   IF Activate = CmdResponseType.CommandActivated THEN
	 CASE Axis OF
		AxisSelectType.Az:
			IF Management.ErrorStatus.errAzimuth=0 THEN
				b_activate_Az:=1;
				b_deactivate_Az:=0;
			ELSE 
				Activate := CmdResponseType.CommandFailed;
			END_IF
		AxisSelectType.El:
			IF Management.ErrorStatus.errElevation=0 THEN
				 b_activate_el:=1;
				 b_deactivate_El:=0;
			ELSE 
				Activate := CmdResponseType.CommandFailed;
			END_IF;
		AxisSelectType.Fi:
			IF Management.ErrorStatus.errFeedIndexer=0 THEN
				 b_activate_fi:=1;
				 b_deactivate_Fi:=0;
			ELSE 
				Activate := CmdResponseType.CommandFailed;
			END_IF;
		AxisSelectType.AzEl:
			IF Management.ErrorStatus.errAzimuth=0 AND Management.ErrorStatus.errElevation=0  THEN
				b_activate_Az:=1;
				b_deactivate_Az:=0;
				b_activate_el:=1;
				b_deactivate_el:=0;
			//	b_SCC_enable_off:=FALSE;
			//	b_SCC_enable_on:=TRUE; 
			ELSE 
				Activate := CmdResponseType.CommandFailed;
			END_IF;
		ELSE 
			//Activate := CmdResponseType.ParameterOutOfRange;
		END_CASE
   END_IF
ELSE 
	Activate := CmdResponseType.NoCmdAuth;
END_IF
CommandArbiter.Status.AxisSelect:=Axis;
CommandArbiter.Status.LastCmdResponse:=Activate;
END_METHOD

METHOD DeActivate : UINT
VAR_INPUT
	SessionID: UINT;
	Axis: UINT;
END_VAR
VAR_OUTPUT
	
END_VAR
VAR
END_VAR
CASE CommandArbiter.Status.DscCmdAuthority OF                    // Check that corerct user is issueing a command
	LMC: IF SessionID= CommandArbiter.Lmc_ID THEN
			DeActivate:= CmdResponseType.CommandActivated;
         END_IF
			
	EGUI: IF SessionID= CommandArbiter.Egui_ID THEN
			DeActivate:= CmdResponseType.CommandActivated;
          END_IF		
ELSE 
     DeActivate:= CmdResponseType.NoCmdAuth;
     Command_Arbiter_error:=1;	
END_CASE

IF DeActivate = CmdResponseType.CommandActivated THEN       // Check Dish State
	Command_Arbiter_error:=0;
	CASE Management.Status.DscState OF 
		DSCStateType.StartUp:
		 	DeActivate := CmdResponseType.CommandRejected;
		DSCStateType.Standby:
		 	DeActivate := CmdResponseType.CommandActivated;
		DSCStateType.Locked:
		 	DeActivate := CmdResponseType.DishLocked;
		DSCStateType.Stowed:
		 	DeActivate :=CmdResponseType.Stowed;
		DSCStateType.Locked_Stowed:
		 	DeActivate := CmdResponseType.DishLocked; 
		DSCStateType.Activating :
		 	DeActivate := CmdResponseType.CommandActivated;
		DSCStateType.Deactivating :
		 	DeActivate := CmdResponseType.CommandActivated;
		DSCStateType.Standstill :
		 	DeActivate := CmdResponseType.CommandActivated;
		DSCStateType.Stopping :
		 	DeActivate := CmdResponseType.CommandActivated;
		DSCStateType.Slew :
		 	DeActivate := CmdResponseType.CommandActivated;
		DSCStateType.Jog :
		 	DeActivate := CmdResponseType.CommandActivated;
		DSCStateType.Track :
		 	DeActivate := CmdResponseType.CommandActivated;
	END_CASE

   IF DeActivate = CmdResponseType.CommandActivated THEN     //Deactivate Axis
	 CASE Axis OF
		AxisSelectType.Az:
		   		b_deactivate_Az:=1;                      //Ladder logic checks for motion and stops axis before deactivating              				
				b_activate_Az:=0;             
		AxisSelectType.El:
		    	b_deactivate_El:=1;
				b_activate_el:=0;
		AxisSelectType.Fi:
		    	b_deactivate_Fi:=1;
	    		b_activate_fi:=0;
		AxisSelectType.AzEl:
		    	b_deactivate_Az:=1;
				b_deactivate_El:=1;	
				b_activate_Az:=0;
				b_activate_el:=0;
	ELSE 
		DeActivate := CmdResponseType.ParameterOutOfRange;
	END_CASE
   END_IF
ELSE 
   DeActivate:= CmdResponseType.NoCmdAuth;
END_IF
CommandArbiter.Status.LastCmdResponse:=DeActivate;
END_METHOD

METHOD Move2Band : UINT
VAR_INPUT
	SessionID : UINT;
	Band :UINT;
END_VAR
CASE CommandArbiter.Status.DscCmdAuthority OF                    // Check that correct user is issueing a command
	LMC: IF SessionID= CommandArbiter.Lmc_ID THEN
			Move2Band:= CmdResponseType.CommandActivated;
     	 END_IF
			
	EGUI: IF SessionID= CommandArbiter.Egui_ID THEN
			Move2Band:= CmdResponseType.CommandActivated;
    	  END_IF		
ELSE 
     Move2Band:= CmdResponseType.NoCmdAuth;
     Command_Arbiter_error:=1;	
END_CASE

IF Move2Band = CmdResponseType.CommandActivated THEN // Check Dish State to see if move is possible
	Command_Arbiter_error:=0;
	IF  Management.ErrorStatus.errGeneral=0 AND Management.WarningStatus.waMngmnt =0 THEN  
		CASE Management.Status.DscState OF 
			 DscStateType.Locked:        Move2Band:=CmdResponseType.DishLocked;
			 DscStateType.Locked_Stowed: Move2Band:=CmdResponseType.DishLocked;
			 DscStateType.Standstill:    Move2Band:=CmdResponseType.CommandActivated;
		     DscStateType.Standby:       Move2Band:=CmdResponseType.CommandActivated;
			 DscStateType.Stowed:	     Move2Band:=CmdResponseType.CommandActivated;
			 DscStateType.Slew:  		 Move2Band:=CmdResponseType.CommandActivated;
			 DscStateType.Track:  		 Move2Band:=CmdResponseType.CommandActivated;
			 DscStateType.Activating:	 Move2Band:=CmdResponseType.CommandActivated;
			 DscStateType.Deactivating:	 Move2Band:=CmdResponseType.CommandActivated;
			 DscStateType.Stopping:		 Move2Band:=CmdResponseType.CommandActivated;
			
		ELSE
		     Move2Band:=CmdResponseType.CommandRejected;
		     Command_Arbiter_error:=1;
		END_CASE	
   		CASE Band OF   // get band position
	 		Bandtype.Optical: r_goto_Fi := LREAL_TO_REAL(gc_r_band_optical - r_pos_fi_v); 
                              FeedIndexer.Status.p_Set:= gc_r_band_optical;   
     		Bandtype.Band_1:  r_goto_Fi := LREAL_TO_REAL(gc_r_band_1 - r_pos_fi_v);
							  FeedIndexer.Status.p_Set:= gc_r_band_1;   
	 		Bandtype.Band_2:  r_goto_Fi := LREAL_TO_REAL(gc_r_band_2 - r_pos_fi_v);
							  FeedIndexer.Status.p_Set:= gc_r_band_2;   
	 		Bandtype.Band_3:  r_goto_Fi := LREAL_TO_REAL(gc_r_band_3 - r_pos_fi_v);
						      FeedIndexer.Status.p_Set:= gc_r_band_3;   
	 		Bandtype.Band_4:  r_goto_Fi := LREAL_TO_REAL(gc_r_band_4 - r_pos_fi_v);
							  FeedIndexer.Status.p_Set:= gc_r_band_4;   
	 		Bandtype.Band_5a: r_goto_Fi := LREAL_TO_REAL(gc_r_band_5a - r_pos_fi_v);
							  FeedIndexer.Status.p_Set:= gc_r_band_5a;   
	 		Bandtype.Band_5b: r_goto_Fi := LREAL_TO_REAL(gc_r_band_5b - r_pos_fi_v);
							  FeedIndexer.Status.p_Set:= gc_r_band_5b;   
	 		Bandtype.Band_6:  r_goto_Fi := LREAL_TO_REAL(gc_r_band_6 - r_pos_fi_v);
							  FeedIndexer.Status.p_Set:= gc_r_band_6;
;   
		END_CASE
	
		IF Move2Band = CmdResponseType.CommandActivated THEN  
			b_activate_Fi:=1;
			b_deactivate_Fi:=0;
			r_goto_v_Fi:= r_vel_max_Fi; 
			b_stop_Fi:= FALSE;
			b_start_goto_Fi:= TRUE;
			b_Move2Band_deactivate:= TRUE;
			Move2Band:=CmdResponseType.CommandActivated;
		ELSE 
			Move2Band:=CmdResponseType.ParameterOutOfRange;
		END_IF             			
							
	ELSE
		Move2Band:=CmdResponseType.CommandRejected;
		Command_Arbiter_error:=1;
	END_IF
END_IF

						

CommandArbiter.Status.LastCmdResponse:=Move2Band;
END_METHOD

METHOD Reset : UINT
VAR_INPUT
	SessionID: UINT;
	Axis: UINT;
END_VAR

VAR
	
END_VAR
CASE CommandArbiter.Status.DscCmdAuthority OF                    // Check that corerct user is issueing a command
	LMC: IF SessionID= CommandArbiter.Lmc_ID THEN
			Reset:= CmdResponseType.CommandActivated;
     	 END_IF
			
	EGUI: IF SessionID= CommandArbiter.Egui_ID THEN
			Reset:= CmdResponseType.CommandActivated;
    	  END_IF		
ELSE 
     Reset:= CmdResponseType.NoCmdAuth;
     Command_Arbiter_error:=1;	
END_CASE

IF Reset = CmdResponseType.CommandActivated THEN
	Command_Arbiter_error:=0;
	CASE Management.Status.DscState OF 
		DSCStateType.StartUp:
		 	Reset := CmdResponseType.CommandActivated;
		DSCStateType.Standby:
		 	Reset := CmdResponseType.CommandActivated;
		DSCStateType.Locked:
		 	Reset := CmdResponseType.CommandActivated;
		DSCStateType.Stowed:
		 	Reset :=CmdResponseType.CommandActivated;
		DSCStateType.Locked_Stowed:
		 	Reset := CmdResponseType.CommandActivated;
		DSCStateType.Activating :
		 	Reset := CmdResponseType.CommandRejected;
		DSCStateType.Deactivating :
		 	Reset := CmdResponseType.CommandRejected;
		DSCStateType.Standstill :
		 	Reset := CmdResponseType.CommandRejected;
		DSCStateType.Stopping :
		 	Reset := CmdResponseType.CommandRejected;
		DSCStateType.Slew :
		 	Reset := CmdResponseType.CommandRejected;
		DSCStateType.Jog :
		 	Reset := CmdResponseType.CommandRejected;
		DSCStateType.Track :
		 	Reset := CmdResponseType.CommandRejected;
	END_CASE

	IF Reset = CmdResponseType.CommandActivated THEN
		CASE Axis OF
			AxisSelectType.Az: b_clear_err_Az:= 1;
			AxisSelectType.El: b_clear_err_El:= 1;
			AxisSelectType.Fi: b_clear_err_Fi:= 1;
			AxisSelectType.AzEl: b_clear_err_Az:= 1;
								 b_clear_err_El:= 1;
			AxisSelectType.Unknown: b_clear_err:= 1;
		ELSE
			Reset := CmdResponseType.ParameterOutOfRange;
		END_CASE
	END_IF 
ELSE 
	 Reset:= CmdResponseType.NoCmdAuth;

END_IF

CommandArbiter.Status.LastCmdResponse:=Reset;
END_METHOD

METHOD SetOnSourceThreshold : Uint
VAR_INPUT
	SessionID :UINT;
	OnSourceThreshold : LREAL;
    ThresholdTimePeriod : LREAL;
END_VAR
CASE CommandArbiter.Status.DscCmdAuthority OF                    // Check that corerct user is issueing a command
	LMC: IF SessionID= CommandArbiter.Lmc_ID THEN
			SetOnSourceThreshold:= CmdResponseType.CommandActivated;
     	 END_IF
			
	EGUI: IF SessionID= CommandArbiter.Egui_ID THEN
			SetOnSourceThreshold:= CmdResponseType.CommandActivated;
    	  END_IF		
ELSE 
     SetOnSourceThreshold:= CmdResponseType.NoCmdAuth;
     Command_Arbiter_error:=1;	
END_CASE

IF SetOnSourceThreshold = CmdResponseType.CommandActivated THEN
	IF (OnSourceThreshold > 0 AND Onsourcethreshold <=20) OR ( ThresholdTimePeriod > 0 AND ThresholdTimePeriod <=10) THEN
		Tracking.Status.OnSourceThreshold:= OnSourceThreshold;
		Tracking.Status.ThresholdTimePeriod:=ThresholdTimePeriod;
		 t_onsource_dev_filt:=LREAL_TO_TIME(ThresholdTimePeriod*1000);
	    command_Arbiter_error:=0;
	ELSE
		SetOnSourceThreshold:= CmdResponseType.ParameterOutOfRange;
		Command_Arbiter_error:=1;
	END_IF
	
ELSE 
	 SetOnSourceThreshold:= CmdResponseType.CommandFailed;
	  Command_Arbiter_error:=1;
END_IF

CommandArbiter.Status.LastCmdResponse:=SetOnSourceThreshold;
END_METHOD

METHOD SetPowerMode : UINT (* Command to set the power mode *)
VAR_INPUT
	SessionID: UINT; (*Seesion ID*)
    LowPowerOn: BOOL:= FALSE; (* True = Low Power mode On *)
    PowerLimKw: LREAL:=10; (* Maximum Power limit in High power Mode *)

END_VAR
CASE CommandArbiter.Status.DscCmdAuthority OF                    // Check that correct user is issueing a command
	LMC: IF SessionID= CommandArbiter.Lmc_ID THEN
			SetPowerMode:= CmdResponseType.CommandActivated;
     	 END_IF
			
	EGUI: IF SessionID= CommandArbiter.Egui_ID THEN
			SetPowerMode:= CmdResponseType.CommandActivated;
    	  END_IF		
ELSE 
     SetPowerMode:= CmdResponseType.NoCmdAuth;
     Command_Arbiter_error:=1;	
END_CASE

IF SetPowerMode = CmdResponseType.CommandActivated THEN       // Check Dish State
	Command_Arbiter_error:=0;
	CASE Management.Status.DscState OF 
		DSCStateType.StartUp:
		 	SetPowerMode := CmdResponseType.CommandRejected;
		DSCStateType.Standby:
		 	SetPowerMode := CmdResponseType.CommandActivated;
		DSCStateType.Locked:
		 	SetPowerMode := CmdResponseType.CommandActivated;
		DSCStateType.Stowed:
		 	SetPowerMode :=CmdResponseType.CommandActivated;
		DSCStateType.Locked_Stowed:
		 	SetPowerMode := CmdResponseType.CommandActivated;
		DSCStateType.Activating :
		 	SetPowerMode := CmdResponseType.CommandActivated;
		DSCStateType.Deactivating :
		 	SetPowerMode := CmdResponseType.CommandActivated;
		DSCStateType.Standstill :
		 	SetPowerMode := CmdResponseType.CommandActivated;
		DSCStateType.Stopping :
		 	SetPowerMode := CmdResponseType.CommandActivated;
		DSCStateType.Slew :
		 	SetPowerMode := CmdResponseType.CommandActivated;
		DSCStateType.Jog :
		 	SetPowerMode := CmdResponseType.CommandActivated;
		DSCStateType.Track :
		 	SetPowerMode := CmdResponseType.CommandActivated;
	END_CASE
END_IF

IF SetPowerMode = CmdResponseType.CommandActivated THEN
	//SetPowerMode := CmdResponseType.NotImplemented;
	IF LowPowerOn =1 THEN 
		Management.PowerStatus.LowPowerActive:=1;
		IF Azimuth.Status.Active THEN
			b_deactivate_Az:=1;
			b_activate_Az:=0;
		END_IF
		
		IF Elevation.Status.Active THEN
			b_deactivate_El:=1;
			b_activate_El:=0;
		END_IF
		
		IF FeedIndexer.Status.Active THEN
			b_deactivate_Fi:=1;
	    	b_activate_Fi:=0;
		END_IF 
					
	ELSE
		Management.PowerStatus.LowPowerActive:=0;
		r_vel_max_Az:=  gc_r_power_Kv_Az*PowerLimKw;
  		r_vel_max_El:=  gc_r_power_Kv_El*PowerLimKw;
  		r_vel_max_Fi:=  gc_r_power_Kv_Fi*PowerLimKw;
		r_goto_acc_Az:= gc_r_power_Ka_Az*PowerLimKw;
  		r_goto_acc_El:= gc_r_power_Ka_El*PowerLimKw;
  		r_goto_acc_Fi:= gc_r_power_Ka_Fi*PowerLimKw;
  	END_IF
END_IF

CommandArbiter.Status.LastCmdResponse:=SetPowerMode;
END_METHOD

METHOD Slew2AbsSingleAx : UINT
VAR_INPUT
	SessionID: UINT;
	Axis: Uint;
	Position:LREAL;
	Speed:LREAL;
END_VAR

VAR
END_VAR
CASE CommandArbiter.Status.DscCmdAuthority OF                    // Check that correct user is issueing a command
	LMC: IF SessionID= CommandArbiter.Lmc_ID THEN
			Slew2AbsSingleAx:= CmdResponseType.CommandActivated;
     	 END_IF
			
	EGUI: IF SessionID= CommandArbiter.Egui_ID THEN
			Slew2AbsSingleAx:= CmdResponseType.CommandActivated;
    	  END_IF		
ELSE 
     Slew2AbsSingleAx:= CmdResponseType.NoCmdAuth;
     Command_Arbiter_error:=1;	
END_CASE

IF Slew2AbsSingleAx = CmdResponseType.CommandActivated THEN // Dish State to see if move is possible
	Command_Arbiter_error:=0;
	//IF  Management.ErrorStatus.errGeneral=0 AND Management.WarningStatus.waMngmnt =0 THEN   If the Dish has errors that prevent movement then it will not be in a state where it can be moved. 
		CASE Management.Status.DscState OF 
			 DscStateType.Locked:        Slew2AbsSingleAx:=CmdResponseType.DishLocked;
			 DscStateType.Locked_Stowed: Slew2AbsSingleAx:=CmdResponseType.DishLocked;
			 DscStateType.Standstill:    Slew2AbsSingleAx:=CmdResponseType.CommandActivated;
		     DscStateType.Standby:       Slew2AbsSingleAx:=CmdResponseType.CommandActivated;
			 DscStateType.Stowed:	     Slew2AbsSingleAx:=CmdResponseType.Stowed;
		ELSE
		     Slew2AbsSingleAx:=CmdResponseType.CommandRejected;
		     Command_Arbiter_error:=1;
		END_CASE								
	//ELSE
	//	Slew2AbsAx:=CmdResponseType.CommandAborted;
	//	Command_Arbiter_error:=1;
	//END_IF
END_IF
	
IF Slew2AbsSingleAx = CmdResponseType.CommandActivated THEN  // Move selected axis
	b_goto_rel:=FALSE;
	CASE Axis OF 
		AxisSelectType.Az:	
            IF (Position <= gc_r_pos_max_Az) AND (Position>= gc_r_pos_min_Az) AND (Speed <= gc_r_vel_max_Az*6) THEN
           		b_activate_Az:=1;
			    r_goto_Az := LREAL_TO_REAL(Position);
				 IF Speed > r_vel_max_Az THEN    // For power management
					 r_goto_v_Az:= r_vel_max_Az;
				 ELSE
				 	 r_goto_v_Az:= LREAL_TO_REAL(Speed/6); 
				 END_IF
				b_stop_Az:= FALSE;
				b_start_goto_Az:= TRUE;
				Slew2AbsSingleAx:=CmdResponseType.CommandActivated;
				r_write_position_az_out:=Position; // Writeing setpoint positions to Cyclic out put to get P.Set outputs
			ELSE 
				Slew2AbsSingleAx:=CmdResponseType.ParameterOutOfRange;
			END_IF			   
		AxisSelectType.El:
 			IF (Position <= gc_r_pos_max_El) AND (Position>= gc_r_pos_min_El) AND (Speed <= gc_r_vel_max_El*6
) THEN
            	b_activate_el:=1;
				r_goto_El := LREAL_TO_REAL(Position);
				
				 IF Speed > r_vel_max_El THEN    // For power management
					 r_goto_v_El:= r_vel_max_El;
				 ELSE
				 	 r_goto_v_El:= LREAL_TO_REAL(Speed/6); 
				 END_IF
				
				b_stop_El:= FALSE;
				b_start_goto_El:= TRUE;
				Slew2AbsSingleAx:=CmdResponseType.CommandActivated;
				r_write_position_el_out:=Position; // Writeing setpoint positions to Cyclic out put to get P.Set outputs
			ELSE 
				Slew2AbsSingleAx:=CmdResponseType.ParameterOutOfRange;
			END_IF 
					    
		AxisSelectType.FI: 
			IF (Position <= gc_r_pos_max_Fi) AND (Position >= gc_r_pos_min_Fi) AND (Speed<= gc_r_vel_max_Fi*6) THEN
                 b_activate_Fi:=1;
				 r_goto_Fi := LREAL_TO_REAL(Position);
				 IF Speed > r_vel_max_Fi THEN 
					 r_goto_v_Fi:= r_vel_max_Fi;
				 ELSE
				 	 r_goto_v_Fi:= LREAL_TO_REAL(Speed/6); 
				 END_IF
				 b_stop_Fi:= FALSE;
				 b_start_goto_Fi:= TRUE;
				 Slew2AbsSingleAx:=CmdResponseType.CommandActivated;
				 r_write_position_fi_out:=Position; // Writeing setpoint positions to Cyclic out put to get P.Set outputs
		    ELSE 
				 Slew2AbsSingleAx:=CmdResponseType.ParameterOutOfRange;
			END_IF              
 			     									
	ELSE
		Slew2AbsSingleAx:=CmdResponseType.ParameterOutOfRange;
	END_CASE
END_IF

CommandArbiter.Status.LastCmdResponse:=Slew2AbsSingleAx;
END_METHOD

METHOD Slew2AbsAzEl : UINT
VAR_INPUT
	SessionID:UINT;
	Pos_Az:LREAL;
	Pos_El:LREAL;
	Speed_Az:LREAL;
	Speed_El:LREAL;
END_VAR
VAR_OUTPUT
	
END_VAR
VAR
	fb_TON: TON;  
	b_flip: BOOL:=False ;
END_VAR
CASE CommandArbiter.Status.DscCmdAuthority OF                    // Check that correct user is issueing a command
	LMC: IF SessionID= CommandArbiter.Lmc_ID THEN
			Slew2AbsAzEl:= CmdResponseType.CommandActivated;
     	 END_IF
			
	EGUI: IF SessionID= CommandArbiter.Egui_ID THEN
			Slew2AbsAzEl:= CmdResponseType.CommandActivated;
    	  END_IF		
ELSE 
     Slew2AbsAzEl:= CmdResponseType.NoCmdAuth;
     Command_Arbiter_error:=1;	
END_CASE

IF Slew2AbsAzEl = CmdResponseType.CommandActivated THEN // Dish State to see if move is possible
	Command_Arbiter_error:=0;
	//IF  Management.ErrorStatus.errGeneral=0 AND Management.WarningStatus.waMngmnt =0 THEN  (*The Dish in the standby state*)
		CASE Management.Status.DscState OF 
			 DscStateType.Locked:        Slew2AbsAzEl:=CmdResponseType.DishLocked;
			 DscStateType.Locked_Stowed: Slew2AbsAzEl:=CmdResponseType.DishLocked;
			 DscStateType.Standstill:    Slew2AbsAzEl:=CmdResponseType.CommandActivated;
		     DscStateType.Standby:       Slew2AbsAzEl:=CmdResponseType.CommandActivated;
			 DscStateType.Stowed:	     Slew2AbsAzEl:=CmdResponseType.Stowed;
			 DscStateType.Slew:          Slew2AbsAzEl:=CmdResponseType.CommandActivated;
		ELSE
		     Slew2AbsAzEl:=CmdResponseType.CommandRejected;
		     Command_Arbiter_error:=1;
		END_CASE								
	(*ELSE
		Slew2AbsAzEl:=CmdResponseType.CommandAborted;
		Command_Arbiter_error:=1;
	END_IF*)
END_IF
	
IF Slew2AbsAzEl = CmdResponseType.CommandActivated THEN  // Move selected axis
	b_goto_rel:=FALSE;
	IF ((Pos_Az <= gc_r_pos_max_Az) AND (Pos_Az >= gc_r_pos_min_Az) AND( Speed_Az <= gc_r_vel_max_Az*6)) AND ((Pos_El <= gc_r_pos_max_El) AND (Pos_El >= gc_r_pos_min_El) AND ( Speed_El <= gc_r_vel_max_El*6)) THEN
		IF b_activate_Az=0 THEN   // Activate axis if it is in Standby
			b_activate_Az:=1;
		END_IF
		IF b_activate_El=0 THEN // Activate axis if it is in Standby
		   b_activate_El:=1;
		END_IF
    		
		r_goto_Az := LREAL_TO_REAL(Pos_Az);
		r_goto_v_Az:= LREAL_TO_REAL(Speed_Az/6); 
		b_stop_Az:= FALSE;
		r_goto_El := LREAL_TO_REAL(Pos_El);
		r_goto_v_El:= LREAL_TO_REAL(Speed_El/6); 
		b_stop_El:= FALSE;
		
		b_slew_az_el:=TRUE;
		
				
		Slew2AbsAzEl:=CmdResponseType.CommandActivated;	
	ELSE 
		Slew2AbsAzEl:=CmdResponseType.ParameterOutOfRange;
	END_IF			   
END_IF
r_write_position_az_out:=Pos_Az; // Writeing setpoint positions to Cyclic out put to get P.Set outputs
r_write_position_el_out:=Pos_El;
CommandArbiter.Status.LastCmdResponse:=Slew2AbsAzEl;
END_METHOD

METHOD Slew2RelSingleAx : UINT
VAR_INPUT
	SessionID:UINT;
	Axis: UINT;
	Position:LREAL;
	Speed:LREAL;
END_VAR
CASE CommandArbiter.Status.DscCmdAuthority OF                    // Check that correct user is issueing a command
	LMC: IF SessionID= CommandArbiter.Lmc_ID THEN
			Slew2RelSingleAx:= CmdResponseType.CommandActivated;
     	 END_IF
			
	EGUI: IF SessionID= CommandArbiter.Egui_ID THEN
			Slew2RelSingleAx:= CmdResponseType.CommandActivated;
    	  END_IF		
ELSE 
     Slew2RelSingleAx:= CmdResponseType.NoCmdAuth;
     Command_Arbiter_error:=1;	
END_CASE

IF Slew2RelSingleAx = CmdResponseType.CommandActivated THEN // Dish State to see if move is possible
	Command_Arbiter_error:=0;
	//IF  Management.ErrorStatus.errGeneral=0 AND Management.WarningStatus.waMngmnt =0 THEN  (*The Dish in the standby state*)
		CASE Management.Status.DscState OF 
			 DscStateType.Locked:        Slew2RelSingleAx:=CmdResponseType.DishLocked;
			 DscStateType.Locked_Stowed: Slew2RelSingleAx:=CmdResponseType.DishLocked;
			 DscStateType.Standstill:    Slew2RelSingleAx:=CmdResponseType.CommandActivated;
		     DscStateType.Standby:       Slew2RelSingleAx:=CmdResponseType.CommandActivated;
			 DscStateType.Stowed:	     Slew2RelSingleAx:=CmdResponseType.Stowed;
		ELSE
		     Slew2RelSingleAx:=CmdResponseType.CommandRejected;
		     Command_Arbiter_error:=1;
		END_CASE								
(*	ELSE
		Slew2RelAx:=CmdResponseType.CommandAborted;
		Command_Arbiter_error:=1;
	END_IF*)
END_IF
	
IF Slew2RelSingleAx = CmdResponseType.CommandActivated THEN  // Move selected axis
	CASE Axis OF 
		AxisSelectType.Az:	
            IF ((Position + r_pos_az_v) <= gc_r_pos_max_Az) AND ((Position + r_pos_az_v )>= gc_r_pos_min_Az) AND ( Speed <= gc_r_vel_max_Az*6) THEN
           		b_activate_Az:=1;
			    r_goto_Az := LREAL_TO_REAL(Position);
				r_goto_v_Az:= LREAL_TO_REAL(Speed/6); 
				b_stop_Az:= FALSE;
				b_start_goto_Az:= TRUE;
				b_goto_rel:=TRUE;
				Slew2RelSingleAx:=CmdResponseType.CommandActivated;
			ELSE 
				Slew2RelSingleAx:=CmdResponseType.ParameterOutOfRange;
			END_IF			   
		AxisSelectType.El:
 			IF ((Position + r_pos_el_v) <= gc_r_pos_max_El) AND ((Position + r_pos_el_v )>= gc_r_pos_min_El) AND ( Speed <= gc_r_vel_max_El*6) THEN
            	b_activate_el:=1;
				r_goto_El := LREAL_TO_REAL(Position);
				r_goto_v_El:= LREAL_TO_REAL(Speed/6); 
				b_stop_El:= FALSE;
				b_start_goto_El:= TRUE;
				b_goto_rel:=TRUE;
				Slew2RelSingleAx:=CmdResponseType.CommandActivated;
			ELSE 
				Slew2RelSingleAx:=CmdResponseType.ParameterOutOfRange;
			END_IF 
					    
		AxisSelectType.FI: 
			IF ((Position + r_pos_fi_v) <= gc_r_pos_max_Fi) AND ((Position + r_pos_fi_v )> gc_r_pos_min_Fi) AND ( Speed <= gc_r_vel_max_Fi*6) THEN
                 b_activate_Fi:=1;
				 r_goto_Fi := LREAL_TO_REAL(Position);
				 r_goto_v_Fi:= LREAL_TO_REAL(Speed/6); 
				 b_stop_Fi:= FALSE;
				 b_start_goto_Fi:= TRUE;
				 b_goto_rel:=TRUE;
				 Slew2RelSingleAx:=CmdResponseType.CommandActivated;
		    ELSE 
				 Slew2RelSingleAx:=CmdResponseType.ParameterOutOfRange;
			END_IF              
 			     									
	ELSE
		Slew2RelSingleAx:=CmdResponseType.ParameterOutOfRange;
	END_CASE
	
		
END_IF
CommandArbiter.Status.AxisSelect:=Axis;
CommandArbiter.Status.LastCmdResponse:=Slew2RelSingleAx;
END_METHOD

METHOD Slew2RelAzEl : UINT
VAR_INPUT
	SessionID:UINT;
	Pos_Az:LREAL;
	Pos_El:LREAL;
	Speed_Az:LREAL;
	Speed_El:LREAL;
	
END_VAR
CASE CommandArbiter.Status.DscCmdAuthority OF                    // Check that correct user is issueing a command
	LMC: IF SessionID= CommandArbiter.Lmc_ID THEN
			Slew2RelAzEl:= CmdResponseType.CommandActivated;
     	 END_IF
			
	EGUI: IF SessionID= CommandArbiter.Egui_ID THEN
			Slew2RelAzEl:= CmdResponseType.CommandActivated;
    	  END_IF		
ELSE 
     Slew2RelAzEl:= CmdResponseType.NoCmdAuth;
     Command_Arbiter_error:=1;	
END_CASE

IF Slew2RelAzEl = CmdResponseType.CommandActivated THEN // Dish State to see if move is possible
	Command_Arbiter_error:=0;
	//IF  Management.ErrorStatus.errGeneral=0 AND Management.WarningStatus.waMngmnt =0 THEN  (*The Dish in the standby state*)
		CASE Management.Status.DscState OF 
			 DscStateType.Locked:        Slew2RelAzEl:=CmdResponseType.DishLocked;
			 DscStateType.Locked_Stowed: Slew2RelAzEl:=CmdResponseType.DishLocked;
			 DscStateType.Standstill:    Slew2RelAzEl:=CmdResponseType.CommandActivated;
		     DscStateType.Standby:       Slew2RelAzEl:=CmdResponseType.CommandActivated;
			 DscStateType.Stowed:	     Slew2RelAzEl:=CmdResponseType.Stowed;
		ELSE
		     Slew2RelAzEl:=CmdResponseType.CommandRejected;
		     Command_Arbiter_error:=1;
		END_CASE								
	(*ELSE
		Slew2RelAzEl:=CmdResponseType.CommandAborted;
		Command_Arbiter_error:=1;
	END_IF *)
END_IF
	
IF Slew2RelAzEl = CmdResponseType.CommandActivated THEN  // Move selected axis
	IF (((Pos_Az + r_pos_az_v) <= gc_r_pos_max_Az) AND ((Pos_Az + r_pos_az_v )>= gc_r_pos_min_Az) AND ( Speed_Az <= gc_r_vel_max_Az*6)) AND (((Pos_El + r_pos_el_v) <= gc_r_pos_max_El) AND ((Pos_El + r_pos_el_v )>= gc_r_pos_min_El) AND ( Speed_El <= gc_r_vel_max_El*6)) THEN
    	b_activate_Az:=1;
		r_goto_Az := LREAL_TO_REAL(Pos_Az);
		b_goto_rel:=TRUE;
		r_goto_v_Az:= LREAL_TO_REAL(Speed_Az/6); 
		b_stop_Az:= FALSE;
		b_start_goto_Az:= TRUE;
		b_activate_el:=1;
		r_goto_El := LREAL_TO_REAL(Pos_El);
		r_goto_v_El:= LREAL_TO_REAL(Speed_El/6); 
		b_stop_El:= FALSE;
		b_start_goto_El:= TRUE;
		Slew2RelAzEl:=CmdResponseType.CommandActivated;	
	ELSE 
		Slew2RelAzEl:=CmdResponseType.ParameterOutOfRange;
	END_IF			   
	
END_IF

CommandArbiter.Status.LastCmdResponse:=Slew2RelAzEl;
END_METHOD

METHOD Stop : UINT
VAR_INPUT
	SessionID:Uint;
	Axis: UINT; 
END_VAR
VAR_OUTPUT
	
END_VAR
VAR
	
END_VAR
CASE CommandArbiter.Status.DscCmdAuthority OF                    // Check that corerct user is issueing a command
	LMC: IF SessionID= CommandArbiter.Lmc_ID THEN
			Stop:= CmdResponseType.CommandActivated;
     	 END_IF
			
	EGUI: IF SessionID= CommandArbiter.Egui_ID THEN
			Stop:= CmdResponseType.CommandActivated;
    	  END_IF		
ELSE 
     Stop:= CmdResponseType.NoCmdAuth;
     Command_Arbiter_error:=1;	
END_CASE

IF Stop = CmdResponseType.CommandActivated THEN
	Command_Arbiter_error:=0;
	CASE Management.Status.DscState OF 
		DSCStateType.StartUp:
		 	Stop := CmdResponseType.CommandRejected;
		DSCStateType.Standby:
		 	Stop := CmdResponseType.CommandRejected;
		DSCStateType.Locked:
		 	Stop := CmdResponseType.DishLocked;
		DSCStateType.Stowed:
		 	Stop :=CmdResponseType.Stowed;
		DSCStateType.Locked_Stowed:
		 	Stop := CmdResponseType.DishLocked; 
		DSCStateType.Activating :
		 	Stop := CmdResponseType.CommandRejected;
		DSCStateType.Deactivating :
		 	Stop := CmdResponseType.CommandRejected;
		DSCStateType.Standstill :
		 	Stop := CmdResponseType.CommandActivated;
		DSCStateType.Stopping :
		 	Stop := CmdResponseType.CommandActivated;
		DSCStateType.Slew :
		 	Stop := CmdResponseType.CommandActivated;
		DSCStateType.Jog :
		 	Stop := CmdResponseType.CommandActivated;
		DSCStateType.Track :
		 	Stop := CmdResponseType.CommandActivated;
	END_CASE

	IF Stop = CmdResponseType.CommandActivated THEN
		b_track_on:=0; // In case a track is runnning then stop the track
		CASE Axis OF
			AxisSelectType.Unknown:  // Stops all 
		       b_scc_stop:=1;
			    b_start_goto_Fi:=0;
			AxisSelectType.Az:
			  b_stop_Az:=1;
			  b_start_goto_Az:=0;
			AxisSelectType.El:
			 b_stop_El:=1;
			 b_start_goto_El:=0;
			AxisSelectType.Fi:
			 b_stop_Fi:=1;
			 b_start_goto_Fi:=0;
			AxisSelectType.AzEl:
			  b_scc_stop:=1;
			   b_stop_Az:=1;
			   b_stop_El:=1;
			   b_start_goto_El:=0;
			   b_start_goto_Az:=0;
		ELSE
			Stop := CmdResponseType.ParameterOutOfRange;
		END_CASE
	END_IF 
			
END_IF
CommandArbiter.Status.LastCmdResponse:= Stop;
END_METHOD

METHOD Stow : Uint
VAR_INPUT
	SessionID:UINT;
	StowAction:BOOL;
END_VAR


VAR
	Speed_El: REAL;
	Speed_Az: Real;
END_VAR
CASE CommandArbiter.Status.DscCmdAuthority OF                    // Check that correct user is issueing a command
	LMC: IF SessionID= CommandArbiter.Lmc_ID THEN
			Stow:= CmdResponseType.CommandActivated;
     	 END_IF
			
	EGUI: IF SessionID= CommandArbiter.Egui_ID THEN
			Stow:= CmdResponseType.CommandActivated;
    	  END_IF		
ELSE 
     Stow:= CmdResponseType.NoCmdAuth;
     Command_Arbiter_error:=1;	
END_CASE

IF Stow = CmdResponseType.CommandActivated THEN // Dish State to see if move is possible
	Command_Arbiter_error:=0;
	IF  Management.ErrorStatus.errGeneral=0 AND Management.WarningStatus.waMngmnt =0 THEN  (*The Dish in the standby state*)
		CASE Management.Status.DscState OF 
			 DscStateType.Locked:        Stow:=CmdResponseType.DishLocked;
			 DscStateType.Locked_Stowed: Stow:=CmdResponseType.DishLocked;
			 DscStateType.Standstill:    Stow:=CmdResponseType.CommandActivated;
		     DscStateType.Standby:       Stow:=CmdResponseType.CommandActivated;
			 DscStateType.Slew:          Stow:=CmdResponseType.CommandActivated;
			 DscStateType.Track:         Stow:=CmdResponseType.CommandActivated;
			                              //Stop Track
			 DscStateType.Stowed:	     Stow:=CmdResponseType.CommandActivated;
		ELSE
		     Stow:=CmdResponseType.CommandRejected;
		     Command_Arbiter_error:=1;
		END_CASE								
	ELSE
		Stow:=CmdResponseType.CommandRejected;
		Command_Arbiter_error:=1;
	END_IF
END_IF

IF Stow = CmdResponseType.CommandActivated THEN
	IF StowAction = TRUE THEN 
		b_activate_Az:=1;
		b_activate_el:=1;
		b_stow:=1; 
		
		IF b_UPS_stow THEN 
		   Speed_Az:= gc_UPS_Stow_Az_Speed;
	       Speed_El:=gc_UPS_Stow_El_Speed; 
		ELSE
		   Speed_Az:= gc_r_vel_max_Az;
	       Speed_El:=gc_r_vel_max_El; 
		END_IF
		
		//r_goto_Az := LREAL_TO_REAL(0-r_pos_az_v);
		r_goto_Az :=0;
		r_goto_v_Az:= LREAL_TO_REAL(Speed_Az); 
		r_goto_El := LREAL_TO_REAL(90-r_pos_el_v);
		r_goto_v_El:= LREAL_TO_REAL(Speed_El); 
		
		
        b_stop_Az:= FALSE;
		//b_start_goto_Az:= TRUE;
		b_stop_El:= FALSE;
		//b_start_goto_El:= TRUE;
		
      // Activates ladder logic A_STOW
		b_stow_pin_retract:=0;	
		
		Stow:=CmdResponseType.CommandActivated;	
	ELSIF StowAction = FALSE THEN 
		b_stow_pin_retract:=1 ;
		//b_stow:= 0;	
	END_IF
END_IF
	
r_write_position_az_out:=0; // Writeing setpoint positions to Cyclic out put to get P.Set outputs
r_write_position_el_out:=90;	

CommandArbiter.Status.LastCmdResponse:=Stow;
END_METHOD

METHOD TrackStartDM : UINT
VAR_INPUT
	SessionID:UINT;
	Interpol :UINT; // 0 = Newton 1= Spline
	StartTime : LREAL ;
	
END_VAR
CASE CommandArbiter.Status.DscCmdAuthority OF                    // Check that corerct user is issueing a command
	LMC: IF SessionID= CommandArbiter.Lmc_ID THEN
			TrackStartDM:= CmdResponseType.CommandActivated;
     	 END_IF
			
	EGUI: IF SessionID= CommandArbiter.Egui_ID THEN
			TrackStartDM:= CmdResponseType.CommandActivated;
    	  END_IF		
ELSE 
     TrackStartDM:= CmdResponseType.NoCmdAuth;
     Command_Arbiter_error:=1;	
END_CASE


IF TrackStartDM = CmdResponseType.CommandActivated THEN // Dish State to see if move is possible
	Command_Arbiter_error:=0;
	IF  Management.ErrorStatus.errGeneral=0 AND Management.WarningStatus.waMngmnt =0 THEN  (*The Dish in the standby state*)
		CASE Management.Status.DscState OF 
			 DscStateType.Locked:        TrackStartDM:=CmdResponseType.DishLocked;
			 DscStateType.Locked_Stowed: TrackStartDM:=CmdResponseType.DishLocked;
			 DscStateType.Standstill:    TrackStartDM:=CmdResponseType.CommandActivated;
		     DscStateType.Standby:       TrackStartDM:=CmdResponseType.CommandActivated;
			 DscStateType.Stowed:	     TrackStartDM:=CmdResponseType.Stowed;
		ELSE
		     TrackStartDM:=CmdResponseType.CommandRejected;
		     Command_Arbiter_error:=1;
		END_CASE								
	ELSE
		TrackStartDM:=CmdResponseType.CommandRejected;
		Command_Arbiter_error:=1;
	END_IF
END_IF


IF TrackStartDM= CmdResponseType.CommandActivated AND(StartTime> Time_cds.Status.TAIoffset) THEN
	TrackStartDM:=CmdResponseType.CommandActivated;	
	b_track_start:=1;
	lr_track_start_time:=StartTime;
ELSIF StartTime < 0 THEN  // Times can't be less than zero
	TrackStartDM:=CmdResponseType.ParameterOutOfRange;
ELSE 	
	TrackStartDM:=CmdResponseType.CommandActivated;	
	b_track_start:=1;
	lr_track_start_time:=Time_cds.Status.TAIoffset+0.1; // add 100ms to give enough time to start track. 
END_IF			   



CommandArbiter.Status.LastCmdResponse:=TrackStartDM;
END_METHOD

METHOD TrackStartPolyDM : UINT
VAR_INPUT
	SessionID: UINT;
	TrackId: UINT; 
	Order : UINT;
		
END_VAR
CASE CommandArbiter.Status.DscCmdAuthority OF                    // Check that corerct user is issueing a command
	LMC: IF SessionID= CommandArbiter.Lmc_ID THEN
			TrackStartPolyDM:= CmdResponseType.CommandActivated;
     	 END_IF
			
	EGUI: IF SessionID= CommandArbiter.Egui_ID THEN
			TrackStartPolyDM:= CmdResponseType.CommandActivated;
    	  END_IF		
ELSE 
    TrackStartPolyDM:= CmdResponseType.NoCmdAuth;
     Command_Arbiter_error:=1;	
END_CASE


TrackStartPolyDM:=CmdResponseType.NotImplemented;
CommandArbiter.Status.LastCmdResponse:=TrackStartPolyDM;
END_METHOD

END_FUNCTION_BLOCK

// IndraMotionMlc1/Application/POUs/OPCUA/OPCUA_Method/fb_Pointing
(*{attribute 'opcua.mapping.type' := ''}
{attribute 'opcua.mapping.modeluri' := 'http://skao.int/DS_ICD/'}
{attribute 'opcua.mapping.publicationdate' := '12/14/2023 00:00:00'}
{attribute 'opcua.mapping.nodeid' := 'nsu=http://skao.int/DS_ICD/;i=1014'}*)
FUNCTION_BLOCK fb_Pointing
VAR_INPUT
	Commands: fb_Pointing_Commands;
	Status: PointingStatus_Type;
	AmbTempParameters: AmbTempParam_Type;
	StaticPmParameters: ARRAY [0..7] OF StaticPmParam;
	TiltmeterParameters: TiltmeterParam;
	
	
	
END_VAR
VAR
	TE :LREAL:=0; 
	
END_VAR

END_FUNCTION_BLOCK

// IndraMotionMlc1/Application/POUs/OPCUA/OPCUA_Method/fb_Pointing_Commands
(*{attribute 'opcua.mapping.type' := ''}
{attribute 'opcua.mapping.modeluri' := 'http://skao.int/DS_ICD/'}
{attribute 'opcua.mapping.publicationdate' := '12/14/2023 00:00:00'}
{attribute 'opcua.mapping.nodeid' := 'nsu=http://skao.int/DS_ICD/;i=1014'}*)
FUNCTION_BLOCK fb_Pointing_Commands
VAR_INPUT
	
END_VAR

METHOD AmbTempCorrSetup : UINT

VAR_INPUT
	SessionID:Uint;
	filt_dt:LREAL;
	ambTempParam1:LREAL;
	ambTempParam2:LREAL;
	ambTempParam3:LREAL;
	ambTempParam4:LREAL;
	ambTempParam5:LREAL;
	ambTempParam6:LREAL;
END_VAR
VAR_OUTPUT
	
END_VAR
VAR
END_VAR
IF SessionID = CommandArbiter.Egui_ID AND CommandArbiter.Status.DscCmdAuthority= EGUI THEN
	Command_Arbiter_error:=0;
	IF filt_dt>=0 AND  filt_dt<=1000 THEN         // Only checks if filt_dt is in range
		Pointing.AmbTempParameters.filt_dt:=filt_dt;
		Pointing.AmbTempParameters.ambTempParam1:=ambTempParam1;
		Pointing.AmbTempParameters.ambTempParam2:=ambTempParam2;
		Pointing.AmbTempParameters.ambTempParam3:=ambTempParam3;
		Pointing.AmbTempParameters.ambTempParam4:=ambTempParam4;
		Pointing.AmbTempParameters.ambTempParam5:=ambTempParam5;
		Pointing.AmbTempParameters.ambTempParam6:=ambTempParam6;	
		AmbTempCorrSetup:=CmdResponseType.CommandDone;
	ELSE
		AmbTempCorrSetup:=CmdResponseType.ParameterOutOfRange;		
	END_IF
ELSE
  AmbTempCorrSetup:=CmdResponseType.NoCmdAuth;
Command_Arbiter_error:=1;	
END_IF

CommandArbiter.Status.LastCmdResponse:= AmbTempCorrSetup;
END_METHOD

METHOD PmCorrOnOff : UINT

VAR_INPUT
	SessionID:UINT;
	StaticOn:BOOL;
	TiltOn:UINT;
	AmbTOn:BOOL;
	Band:UINT;
	
END_VAR
VAR_OUTPUT
	
END_VAR
VAR
END_VAR
CASE CommandArbiter.Status.DscCmdAuthority OF                    // Check that corerct user is issueing a command
	LMC: IF SessionID= CommandArbiter.Lmc_ID THEN
			PmCorrOnOff:= CmdResponseType.CommandActivated;
         END_IF
			
	EGUI: IF SessionID= CommandArbiter.Egui_ID THEN
			PmCorrOnOff:= CmdResponseType.CommandActivated;
     	  END_IF		
ELSE 
     PmCorrOnOff:= CmdResponseType.NoCmdAuth;
     Command_Arbiter_error:=1;	
END_CASE

IF PmCorrOnOff = CmdResponseType.CommandActivated THEN 
	IF  Band <8 AND Band >= 0 THEN 
		Command_Arbiter_error:=0;
		Pointing.Status.BandForCorr:=Band;
		PmCorrOnOff:=CmdResponseType.CommandDone;
		IF StaticOn THEN
	    	Pointing.Status.StaticCorrActive:=TRUE;
		ELSE
			Pointing.Status.StaticCorrActive:=FALSE;		
		END_IF
		
		IF AmbTOn THEN
			Pointing.Status.AmbTempCorrActive:=TRUE;
		ELSE
			Pointing.Status.AmbTempCorrActive:=FALSE;	
		END_IF
	
		CASE TiltOn OF
        	0: Pointing.Status.TiltCorrActive:=0;
			   Pointing.Status.TiltOne_On:=0;
			   Pointing.Status.TiltTwo_On:=0;
						
        	1: Pointing.Status.TiltCorrActive:=1;
		   	   Pointing.Status.TiltOne_On:=1;
			   Pointing.Status.TiltTwo_On:=0;
			   
			2: Pointing.Status.TiltCorrActive:=1;
		   	   Pointing.Status.TiltOne_On:=0;
			   Pointing.Status.TiltTwo_On:=1;
   	 	ELSE
			PmCorrOnOff:=CmdResponseType.ParameterOutOfRange;
		END_CASE
	   
	ELSE 
		PmCorrOnOff:=CmdResponseType.ParameterOutOfRange;
	END_IF
END_IF
CommandArbiter.Status.LastTiltOn:=TiltOn;
CommandArbiter.Status.LastCmdResponse:= PmCorrOnOff;
END_METHOD

METHOD StaticPmSetup : UINT
VAR_INPUT
	SessionID:UINT;
	Band:UINT;
	IA:LREAL;
	CA:LREAL;
	NPAE:LREAL;
	AN:LREAL;
	AN0:LREAL;
	AW:LREAL;
	AW0:LREAL;
	ACEC:LREAL;
	ACES:LREAL;
	ABA:LREAL;
	ABphi:LREAL;
	IE:LREAL;
	ECEC: LREAL;
	ECES: LREAL;
	HECE4: LREAL;
	HESE4:LREAL;
	HECE8:LREAL;
	HESE8:LREAL;

END_VAR
VAR_OUTPUT
	
END_VAR
VAR
END_VAR
CASE CommandArbiter.Status.DscCmdAuthority OF                    // Check that corerct user is issueing a command
	LMC: IF SessionID= CommandArbiter.Lmc_ID THEN
			StaticPmSetup:= CmdResponseType.CommandActivated;
         END_IF
			
	EGUI: IF SessionID= CommandArbiter.Egui_ID THEN
			StaticPmSetup:= CmdResponseType.CommandActivated;
     	  END_IF		
ELSE 
     StaticPmSetup:= CmdResponseType.NoCmdAuth;
     Command_Arbiter_error:=1;	
END_CASE



IF StaticPmSetup = CmdResponseType.CommandActivated  THEN
	Command_Arbiter_error:=0;
	IF Band >=0 AND Band <8 THEN
		Pointing.StaticPmParameters[Band].IA:=IA;
		Pointing.StaticPmParameters[Band].CA:=CA;
		Pointing.StaticPmParameters[Band].NPAE:=NPAE;
		Pointing.StaticPmParameters[Band].AN:=AN;
		Pointing.StaticPmParameters[Band].AN0:=AN0;
		Pointing.StaticPmParameters[Band].AW:=AW;
		Pointing.StaticPmParameters[Band].AW0:=AW0;
		Pointing.StaticPmParameters[Band].ACEC:=ACEC;
		Pointing.StaticPmParameters[Band].ACES:=ACES;
		Pointing.StaticPmParameters[Band].ABA:=ABA;
		Pointing.StaticPmParameters[Band].ABphi:=ABphi;
		Pointing.StaticPmParameters[Band].IE:=IE;
		Pointing.StaticPmParameters[Band].ECEC:=ECEC;
		Pointing.StaticPmParameters[Band].ECES:=ECES;
		Pointing.StaticPmParameters[Band].HECE4:=HECE4;
		Pointing.StaticPmParameters[Band].HESE4:=HESE4;
		Pointing.StaticPmParameters[Band].HECE8:=HECE8;
		Pointing.StaticPmParameters[Band].HESE8:=HESE8;
		StaticPmSetup:=CmdResponseType.CommandDone;
	ELSE
   		StaticPmSetup:=CmdResponseType.ParameterOutOfRange;	
	END_IF
ELSE
   StaticPmSetup:=CmdResponseType.NoCmdAuth;	
   Command_Arbiter_error:=1;
END_IF
CommandArbiter.Status.LastCmdResponse:=StaticPmSetup;
END_METHOD

METHOD TiltCalSetup : UINT
VAR_INPUT
	SessionID:Uint;
	TiltmeterPos:UINT;
	Tiltmeter_serial_no:STRING;
	tilt_temp_scale:LREAL;
	x_filt_dt:LREAL;
	x_off:LREAL;
	x_offTC:LREAL;
	x_scale:LREAL;
	x_scaleTC:LREAL;
	x_zero:LREAL;
	x_zeroTC:LREAL;
	y_filt_dt:LREAL;
	y_off:LREAL;
	y_offTC:LREAL;
	y_scale:LREAL;
	y_scaleTC:LREAL;
	y_zero:LREAL;
	y_zeroTC:LREAL;
	
	
END_VAR
VAR_OUTPUT
	
END_VAR
VAR
END_VAR
IF SessionID = CommandArbiter.Egui_ID AND CommandArbiter.Status.DscCmdAuthority = EGUI THEN
	Command_Arbiter_error:=0;
	IF TiltmeterPos=1  THEN
		Pointing.TiltmeterParameters.One.Tiltmeter_serial_no:=Tiltmeter_serial_no;
		Pointing.TiltmeterParameters.One.Tilt_temp_scale:=Tilt_temp_scale;
		Pointing.TiltmeterParameters.One.x_scale:=x_scale;
		Pointing.TiltmeterParameters.One.x_scaleTC:=x_scaleTC;
		Pointing.TiltmeterParameters.One.x_zero:=x_zero;
		Pointing.TiltmeterParameters.One.x_zeroTC:=x_zeroTC;
		Pointing.TiltmeterParameters.One.x_off:=x_off;
		Pointing.TiltmeterParameters.One.x_offTC:=x_offTC;
		Pointing.TiltmeterParameters.One.x_filt_dt:=x_filt_dt;
		Pointing.TiltmeterParameters.One.y_scale:=y_scale;
		Pointing.TiltmeterParameters.One.y_scaleTC:=y_scaleTC;
		Pointing.TiltmeterParameters.One.y_zero:=y_zero;
		Pointing.TiltmeterParameters.One.y_zeroTC:=y_zeroTC;
		Pointing.TiltmeterParameters.One.y_off:=y_off;
		Pointing.TiltmeterParameters.One.y_offTC:=y_offTC;
		Pointing.TiltmeterParameters.One.y_filt_dt:=y_filt_dt;
		TiltCalSetup:=CmdResponseType.CommandDone;
	ELSIF TiltmeterPos=2  THEN
		Pointing.TiltmeterParameters.Two.Tiltmeter_serial_no:=Tiltmeter_serial_no;
		Pointing.TiltmeterParameters.Two.Tilt_temp_scale:=Tilt_temp_scale;
		Pointing.TiltmeterParameters.Two.x_scale:=x_scale;
		Pointing.TiltmeterParameters.Two.x_scaleTC:=x_scaleTC;
		Pointing.TiltmeterParameters.Two.x_zero:=x_zero;
		Pointing.TiltmeterParameters.Two.x_zeroTC:=x_zeroTC;
		Pointing.TiltmeterParameters.Two.x_off:=x_off;
		Pointing.TiltmeterParameters.Two.x_offTC:=x_offTC;
		Pointing.TiltmeterParameters.Two.x_filt_dt:=x_filt_dt;
		Pointing.TiltmeterParameters.Two.y_scale:=y_scale;
		Pointing.TiltmeterParameters.Two.y_scaleTC:=y_scaleTC;
		Pointing.TiltmeterParameters.Two.y_zero:=y_zero;
		Pointing.TiltmeterParameters.Two.y_zeroTC:=y_zeroTC;
		Pointing.TiltmeterParameters.Two.y_off:=y_off;
		Pointing.TiltmeterParameters.Two.y_offTC:=y_offTC;
		Pointing.TiltmeterParameters.Two.y_filt_dt:=y_filt_dt;
		TiltCalSetup:=CmdResponseType.CommandDone;	
	ELSE
		TiltCalSetup:=CmdResponseType.ParameterOutOfRange;		
	END_IF
ELSE
   TiltCalSetup:=CmdResponseType.NoCmdAuth;	
   Command_Arbiter_error:=1;
END_IF

CommandArbiter.Status.LastCmdResponse:=TiltCalSetup;
END_METHOD

END_FUNCTION_BLOCK

// IndraMotionMlc1/Application/POUs/OPCUA/OPCUA_Method/fb_Safety
(*{attribute 'opcua.mapping.type' := ''}
{attribute 'opcua.mapping.modeluri' := 'http://skao.int/DS_ICD/'}
{attribute 'opcua.mapping.publicationdate' := '12/14/2023 00:00:00'}
{attribute 'opcua.mapping.nodeid' := 'nsu=http://skao.int/DS_ICD/;i=1012'}*)
FUNCTION_BLOCK fb_Safety
VAR_INPUT	
	Commands: fb_Safety_Commands;
	Status: SafetyStatus_Type;
	
END_VAR

END_FUNCTION_BLOCK

// IndraMotionMlc1/Application/POUs/OPCUA/OPCUA_Method/fb_Safety_Commands
(*{attribute 'opcua.mapping.type' := ''}
{attribute 'opcua.mapping.modeluri' := 'http://skao.int/DS_ICD/'}
{attribute 'opcua.mapping.publicationdate' := '12/14/2023 00:00:00'}
{attribute 'opcua.mapping.nodeid' := 'nsu=http://skao.int/DS_ICD/;i=1012'}*)
FUNCTION_BLOCK fb_Safety_Commands
VAR_INPUT	
	
	
END_VAR

METHOD InterlockAck :UINT
VAR_INPUT
	SessionID:UINT;	
END_VAR
VAR_OUTPUT
	
END_VAR
VAR
	b_clear_interlock:BOOL;
	
END_VAR
CASE CommandArbiter.Status.DscCmdAuthority OF                    // Check that corerct user is issueing a command
	LMC: IF SessionID = CommandArbiter.Lmc_ID THEN
			InterlockAck:= CmdResponseType.CommandActivated;
         END_IF
			
	EGUI: IF SessionID = CommandArbiter.Egui_ID THEN
		     InterlockAck:= CmdResponseType.CommandActivated;
          END_IF		
ELSE 
     InterlockAck:= CmdResponseType.NoCmdAuth;
     Command_Arbiter_error:=1;	
END_CASE

IF InterlockAck = CmdResponseType.CommandActivated THEN     // Check if the Command can be used in the current dish state
	CASE Management.Status.DscState OF 
		DSCStateType.Locked:
		 	InterlockAck := CmdResponseType.CommandActivated;
		DSCStateType.Locked_Stowed:
		 	InterlockAck := CmdResponseType.CommandActivated;
	ELSE
		InterlockAck := CmdResponseType.CommandFailed;
		Command_Arbiter_error:=1;	
	END_CASE
END_IF

IF InterlockAck = CmdResponseType.CommandActivated THEN   // Clear the interlocks
	Command_Arbiter_error:=0;
  IF  Safety.Status.InterlockClearable THEN
	//b_clear_interlock:=1;
	b_Estop_active:=0;
	b_interlock_active_Az:=0;
	b_interlock_active_El:=0;
	b_interlock_active_Fi:=0;
	Safety.Status.InterlockClearable:=0;
	InterlockAck:=CmdResponseType.CommandDone;		
  ELSE 
	InterlockAck:=CmdResponseType.CommandRejected;
	b_clear_interlock:=0;
  END_IF
END_IF

CommandArbiter.Status.LastCmdResponse:= InterlockAck;
END_METHOD

METHOD MoveStowPin :UINT
VAR_INPUT	
	SessionID: UINT;
	StowPinDeploy:BOOL;
END_VAR
	
VAR_OUTPUT
	
END_VAR
VAR
	Users:STRING;
END_VAR
CASE CommandArbiter.Status.DscCmdAuthority OF                    // Check that corerct user is issueing a command
		
	EGUI: IF SessionID = CommandArbiter.Egui_ID THEN
		     MoveStowPin:= CmdResponseType.CommandActivated;
          ELSE 
			 MoveStowPin:= CmdResponseType.NoCmdAuth;
		  END_IF		
ELSE 
     MoveStowPin:= CmdResponseType.NoCmdAuth;
     Command_Arbiter_error:=1;	
END_CASE

IF MoveStowPin = CmdResponseType.CommandActivated THEN     // Check if the Command can be used in the current dish state
	CASE Management.Status.DscState OF 
		DscStateType.StartUp:
		    MoveStowPin := CmdResponseType.CommandActivated;
		DscStateType.Standstill:
		    MoveStowPin := CmdResponseType.CommandActivated;
		DscStateType.Standby :
			MoveStowPin := CmdResponseType.CommandActivated;
		DSCStateType.Locked:
		 	MoveStowPin := CmdResponseType.DishLocked;
		DSCStateType.Locked_Stowed:
		 	MoveStowPin := CmdResponseType.DishLocked;
		DSCStateType.Stowed	:
		    MoveStowPin := CmdResponseType.CommandActivated;
	ELSE
		MoveStowPin := CmdResponseType.CommandFailed;
		Command_Arbiter_error:=1;	
	END_CASE

END_IF

IF MoveStowPin = CmdResponseType.CommandActivated AND b_stow_lock_allow THEN  // Check that Azimuth is in the correct position 
	Command_Arbiter_error:=0;
			IF StowPinDeploy= TRUE THEN
				IF b_stow_pin_limit_lock  THEN
					MoveStowPin:=CmdResponseType.Stowed;
				ELSE
					b_manual_stow:=1;
					MoveStowPin:=CmdResponseType.CommandActivated;
				END_IF		
			END_IF
	
ELSIF MoveStowPin = CmdResponseType.CommandActivated AND StowPinDeploy= FALSE THEN //Need to be able to retract Stow pin even if Encoders are in incorrect position 
	IF b_stow_pin_limit_unlock  THEN
		MoveStowPin:=CmdResponseType.CommandDone;
	ELSE
		b_manual_stow:=0;
		b_stow_pin_retract:=1;
		MoveStowPin:=CmdResponseType.CommandActivated;
	END_IF		
ELSE 
    MoveStowPin:=CmdResponseType.CommandFailed;			
END_IF		
CommandArbiter.Status.LastCmdResponse:=MoveStowPin;
END_METHOD

END_FUNCTION_BLOCK

// IndraMotionMlc1/Application/POUs/OPCUA/OPCUA_Method/fb_Time_cds
(*{attribute 'opcua.mapping.type' := ''}
{attribute 'opcua.mapping.modeluri' := 'http://skao.int/DS_ICD/'}
{attribute 'opcua.mapping.publicationdate' := '12/14/2023 00:00:00'}
{attribute 'opcua.mapping.nodeid' := 'nsu=http://skao.int/DS_ICD/;i=1023'}*)
FUNCTION_BLOCK fb_Time_cds
VAR_INPUT
	Commands: fb_Time_Commands;
	Status : Time_cdsStatus_Type;
	
END_VAR

END_FUNCTION_BLOCK

// IndraMotionMlc1/Application/POUs/OPCUA/OPCUA_Method/fb_Time_Commands
(*{attribute 'opcua.mapping.type' := ''}
{attribute 'opcua.mapping.modeluri' := 'http://skao.int/DS_ICD/'}
{attribute 'opcua.mapping.publicationdate' := '12/14/2023 00:00:00'}
{attribute 'opcua.mapping.nodeid' := 'nsu=http://skao.int/DS_ICD/;i=1023'}*)
FUNCTION_BLOCK fb_Time_Commands
VAR_INPUT
	
END_VAR

METHOD SetTimeSource : UINT
VAR_INPUT
	SessionID:  UINT;
	DscTimeSyncSource:UINT;
	TimeSourceAddrNTP:STRING;
END_VAR
VAR_OUTPUT
	
END_VAR
IF SessionID = CommandArbiter.Egui_ID AND CommandArbiter.Status.DscCmdAuthority = EGUI THEN
	Command_Arbiter_error:=0;
	CASE DscTimeSyncSource OF 
		DscTimeSyncSourceType.DSC:
			Time_cds.Status.DscTimeSyncSource:= DscTimeSyncSourceType.DSC;
			Source_Timesync:=2;
			SetTimeSource:=CmdResponseType.CommandActivated;
		DscTimeSyncSourceType.NTP:
		    Time_cds.Status.DscTimeSyncSource:= DscTimeSyncSourceType.NTP;
			Source_Timesync:=1;
			IP_Adress_NTP:=TimeSourceAddrNTP;
			SetTimeSource:=CmdResponseType.CommandActivated;
			b_ntp_update_start:=TRUE;
			
		DscTimeSyncSourceType.PTP:
			Time_cds.Status.DscTimeSyncSource:= DscTimeSyncSourceType.PTP;
			Source_Timesync:=0;
			IP_Adress_PTP:=TimeSourceAddrNTP;
			SetTimeSource:=CmdResponseType.CommandActivated;
     ELSE
		 SetTimeSource:=CmdResponseType.ParameterOutOfRange;
	END_CASE
ELSE
   SetTimeSource:=CmdResponseType.NoCmdAuth;
   Command_Arbiter_error:=1;	
END_IF

CommandArbiter.Status.LastCmdResponse:= SetTimeSource;
END_METHOD

END_FUNCTION_BLOCK

// IndraMotionMlc1/Application/POUs/OPCUA/OPCUA_Method/fb_Tracking
(*{attribute 'opcua.mapping.type' := ''}
{attribute 'opcua.mapping.modeluri' := 'http://skao.int/DS_ICD/'}
{attribute 'opcua.mapping.publicationdate' := '12/14/2023 00:00:00'}
{attribute 'opcua.mapping.nodeid' := 'nsu=http://skao.int/DS_ICD/;i=1036'}*)
FUNCTION_BLOCK fb_Tracking
VAR_INPUT
	Commands: fb_Tracking_Commands; 
	Status : TrackingStatus_Type;
	PolyStatus: PolyStatus_type;
	TableStatus: TableStatus_type;
END_VAR

END_FUNCTION_BLOCK

// IndraMotionMlc1/Application/POUs/OPCUA/OPCUA_Method/fb_Tracking_Commands
(*{attribute 'opcua.mapping.type' := ''}
{attribute 'opcua.mapping.modeluri' := 'http://skao.int/DS_ICD/'}
{attribute 'opcua.mapping.publicationdate' := '12/14/2023 00:00:00'}
{attribute 'opcua.mapping.nodeid' := 'nsu=http://skao.int/DS_ICD/;i=1036'}*)
FUNCTION_BLOCK fb_Tracking_Commands
VAR

END_VAR

METHOD TrackLoadStaticOff : Uint
VAR_INPUT
	SessionID:UINT;
	Off_Xel : LREAL;
	Off_El: LREAL;
	
END_VAR
CASE CommandArbiter.Status.DscCmdAuthority OF                    // Check that corerct user is issueing a command
	LMC: IF SessionID= CommandArbiter.Lmc_ID THEN
			TrackLoadStaticOff:= CmdResponseType.CommandActivated;
     	 END_IF
			
	EGUI: IF SessionID= CommandArbiter.Egui_ID THEN
			TrackLoadStaticOff:= CmdResponseType.CommandActivated;
    	  END_IF		
ELSE 
     TrackLoadStaticOff:= CmdResponseType.NoCmdAuth;
     Command_Arbiter_error:=1;	
END_CASE

IF TrackLoadStaticOff = CmdResponseType.CommandActivated THEN 
	IF ABS(Off_El)<= gc_r_El_off_limit AND ABS(Off_Xel)<= gc_r_Xel_off_limit THEN 
	tracking.Status.act_statOffset_value_El:=Off_El;
	tracking.Status.act_statOffset_value_Xel:=Off_Xel;
	ELSE 
		TrackLoadStaticOff:= CmdResponseType.ParameterOutOfRange;
	END_IF
END_IF

CommandArbiter.Status.LastCmdResponse:= TrackLoadStaticOff;
END_METHOD

METHOD TrackLoadTable : UINT
VAR_INPUT
	SessionID:UINT;
	LoadMode :UINT;
	SequenceLength :UINT;
    TaiOffset: ARRAY [1..1000] OF LREAL;
	Azimuth: ARRAY [1..1000] OF LREAL;
	Elevation: ARRAY [1..1000] OF LREAL;
END_VAR

VAR
 i: UINT:=1 ;
 index: UINT:=1 ;
 ValidStart: UINT:=0 ;
END_VAR

CASE CommandArbiter.Status.DscCmdAuthority OF                    // Check that corerct user is issueing a command
	LMC: IF SessionID= CommandArbiter.Lmc_ID THEN
			TrackLoadTable:= CmdResponseType.CommandActivated;
     	 END_IF
			
	EGUI: IF SessionID= CommandArbiter.Egui_ID THEN
			TrackLoadTable:= CmdResponseType.CommandActivated;
    	  END_IF		
ELSE 
     TrackLoadTable:= CmdResponseType.NoCmdAuth;
     Command_Arbiter_error:=1;	
END_CASE

IF TrackLoadTable = CmdResponseType.CommandActivated THEN 
  	IF LoadMode=0 AND(10000-i_num_stack_left) < Sequencelength THEN // Check that there is enough space in the stack.
		TrackLoadTable:= CmdResponseType.CommandFailed;
		
	ELSIF LoadMode=0 AND TaiOffset[SequenceLength] < track_table[i_End].TAIoffset THEN // Check if any point in the loaded table is at the end of the table
		TrackLoadTable:= CmdResponseType.ParameterOutOfRange;
		
	ELSE 
		FOR i:= 1 TO (SequenceLength-1) BY 1 DO    // Check that the time is monotonic 
			IF TaiOffset[i]> (TaiOffset[i+1]) THEN   
				TrackLoadTable:= CmdResponseType.NoOfParametersError;
			END_IF
		END_FOR

		FOR i:= 1 TO SequenceLength BY 1 DO  // Check that the positions are within limits
			IF ((Azimuth[i] > gc_r_pos_max_Az) OR (Azimuth[i] < gc_r_pos_min_Az)) OR ((Elevation[i] > gc_r_pos_max_El) OR (Elevation[i] < gc_r_pos_min_El)) THEN 
				TrackLoadTable:= CmdResponseType.ParameterOutOfRange;
			END_IF
		END_FOR
				
		FOR i:=(SequenceLength-1) TO 1 BY -1 DO    // Check for the time in the Sequence when the future time starts
			IF Time_cds.Status.TAIoffset < (TaiOffset[i+1]+0.1) THEN   
				ValidStart:=i;
			END_IF
		END_FOR
		IF ValidStart < 1 THEN    // Check that table has points in the future 
			TrackLoadTable:= CmdResponseType.ParameterOutOfRange;
		END_IF
	END_IF
END_IF

IF TrackLoadTable = CmdResponseType.CommandActivated THEN 
	CASE LoadMode OF
		  
		0: FOR index:= ValidStart TO SequenceLength BY 1 DO  //Append 
			 IF track_table[i_End].TAIoffset<>0 THEN 
				i_End:=F_I_number(i_End+1);
			 END_IF
			 track_table[i_End].TAIoffset:=TaiOffset[index];
			 track_table[i_End].Azimuth:= Azimuth[index];
			 track_table[i_End].Elevation:= Elevation[index];
			 
		   END_FOR  
           CommandArbiter.Status.LastLoadMode:= LoadMode; 
           
		   
		1:  i_End:= i_Start+1;  // Set the end of the table to the Start to over write the points. 
		                        // Consider adding a blend between the different tables. 
			FOR index:= ValidStart TO SequenceLength BY 1 DO  //New 
			  IF track_table[i_End].TAIoffset<>0 THEN
				 i_End:=F_I_number(i_End+1);
			  END_IF
			  track_table[i_End].TAIoffset:=TaiOffset[index];
			  track_table[i_End].Azimuth:= Azimuth[index];
			  track_table[i_End].Elevation:= Elevation[index];
		    END_FOR            
		   CommandArbiter.Status.LastLoadMode:= LoadMode; 
	       
		2:  i_Start:=1;       // Reset to 1st position of the stack. 
            i_End:= i_Start;  // Set the end of the table to the Start to over write the points. 
		                        // Consider adding a blend between the different tables. 
			FOR index:= ValidStart TO SequenceLength BY 1 DO  //New 
			  IF track_table[i_End].TAIoffset<>0 THEN
				 i_End:=F_I_number(i_End+1);
			  END_IF
			  track_table[i_End].TAIoffset:=TaiOffset[index];
			  track_table[i_End].Azimuth:= Azimuth[index];
			  track_table[i_End].Elevation:= Elevation[index];
		    END_FOR            
	           
	END_CASE;
	TrackLoadTable:= CmdResponseType.CommandActivated; // Reset
	CommandArbiter.Status.LastLoadMode:=LoadMode; 
	Tracking.TableStatus.pts_DataValid:=TRUE;
END_IF;

CommandArbiter.Status.LastCmdResponse:= TrackLoadTable;
END_METHOD

METHOD TrackStart :Uint
VAR_INPUT
	SessionID:UINT;
	Interpol:UINT;
	StartTime:LREAL;
END_VAR
VAR_OUTPUT
	
END_VAR
VAR
	
END_VAR
CASE CommandArbiter.Status.DscCmdAuthority OF                    // Check that corerct user is issueing a command
	LMC: IF SessionID= CommandArbiter.Lmc_ID THEN
			TrackStart:= CmdResponseType.CommandActivated;
     	 END_IF
			
	EGUI: IF SessionID= CommandArbiter.Egui_ID THEN
			TrackStart:= CmdResponseType.CommandActivated;
    	  END_IF		
ELSE 
     TrackStart:= CmdResponseType.NoCmdAuth;
     Command_Arbiter_error:=1;	
END_CASE

IF TrackStart = CmdResponseType.CommandActivated THEN // Dish State to see if move is possible
	Command_Arbiter_error:=0;
	IF  Management.ErrorStatus.errGeneral=0 AND Management.WarningStatus.waMngmnt =0 THEN  (*The Dish in the standby state*)
		CASE Management.Status.DscState OF 
			 DscStateType.Locked:        TrackStart:=CmdResponseType.DishLocked;
			 DscStateType.Locked_Stowed: TrackStart:=CmdResponseType.DishLocked;
			 DscStateType.Standstill:    TrackStart:=CmdResponseType.CommandActivated;
		     DscStateType.Standby:       TrackStart:=CmdResponseType.CommandActivated;
			 DscStateType.Stowed:	     TrackStart:=CmdResponseType.Stowed;
			 DscStateType.Track:         TrackStart:=CmdResponseType.CommandActivated;
		ELSE
		     TrackStart:=CmdResponseType.CommandRejected;
		     Command_Arbiter_error:=1;
		END_CASE								
	ELSE
		TrackStart:=CmdResponseType.CommandRejected;
		Command_Arbiter_error:=1;
	END_IF
END_IF
	
IF TrackStart=CmdResponseType.CommandActivated THEN
	IF StartTime > Time_cds.Status.TAIoffset THEN
		b_activate_Az:=1;
		b_activate_El:=1;	
		b_track_start:=1;
		lr_track_start_time:=StartTime;
	ELSIF StartTime < Time_cds.Status.TAIoffset THEN  // Will start tracking immediately
		b_activate_Az:=1;
		b_activate_El:=1;	
		b_track_start:=1;
		lr_track_start_time:=Time_cds.Status.TAIoffset;
	ELSIF StartTime < 0 THEN 
		TrackStart:=CmdResponseType.ParameterOutOfRange;
	ELSE 	
	//	TrackStart:=CmdResponseType.CommandActivated;
	//	b_activate_Az:=1;
	//	b_activate_El:=1;	
    //b_track_start:=1;
	//	lr_track_start_time:=Time_cds.Status.TAIoffset+0.1; // add 100ms to give enough time to start track. 
	END_IF			   
END_IF

Tracking.TableStatus.pts_Interpol:= Interpol;
CommandArbiter.Status.LastCmdResponse:=TrackStart;
END_METHOD

METHOD TrackStartPoly : UINT

VAR_INPUT
	SessionID:UINT;
	TrackId:  UINT;
	Order : UINT;
END_VAR

VAR
	
END_VAR
// Check Auth
// Check parameters
// Check State
TrackStartPoly := CmdResponseType.NotImplemented;

CommandArbiter.Status.LastCmdResponse:=TrackStartPoly;
END_METHOD

END_FUNCTION_BLOCK

// IndraMotionMlc1/Application/POUs/Panel Function/DANCE_OFF
PROGRAM DANCE_OFF
VAR
	R_TRIG_0: R_TRIG;
	dance_enable: BOOL;
	R_TRIG_1: R_TRIG;
	MC_Power_0: MC_Power;
	MC_MoveAbsolute_0: MC_MoveAbsolute;
	R_TRIG_2: R_TRIG;
	MC_MoveAbsolute_1: MC_MoveAbsolute;
	R_TRIG_3: R_TRIG;
	MC_MoveAbsolute_2: MC_MoveAbsolute;
	R_TRIG_4: R_TRIG;
	dance_step1: BOOL;
	MC_MoveAbsolute_3: MC_MoveAbsolute;
	R_TRIG_5: R_TRIG;
	dance_step2: BOOL;
	MC_MoveAbsolute_4: MC_MoveAbsolute;
	R_TRIG_6: R_TRIG;
	TON_0: TON;
	R_TRIG_7: R_TRIG;
	TON_1: TON;
	dance_step3: BOOL;
	TON_2: TON;
	dance_step4: BOOL;
	MC_MoveAbsolute_5: MC_MoveAbsolute;
	R_TRIG_8: R_TRIG;
	TON_3: TON;
	dance_step5: BOOL;
	MC_MoveAbsolute_6: MC_MoveAbsolute;
	R_TRIG_9: R_TRIG;
	TON_4: TON;
	dance_step6: BOOL;
	MC_MoveAbsolute_7: MC_MoveAbsolute;
	R_TRIG_10: R_TRIG;
	TON_5: TON;
	dance_step7: BOOL;
	R_TRIG_11: R_TRIG;
	dance_step8: BOOL;
	MC_MoveAbsolute_8: MC_MoveAbsolute;
	R_TRIG_12: R_TRIG;
	TON_6: TON;
	F_TRIG_0: F_TRIG;
	TON_7: TON;
	R_TRIG_13: R_TRIG;
	dance_step9: BOOL;
	R_TRIG_14: R_TRIG;
	TON_8: TON;
	TON_9: TON;
	R_TRIG_15: R_TRIG;
	TON_10: TON;
	dance_step10: BOOL;
	TON_11: TON;
END_VAR

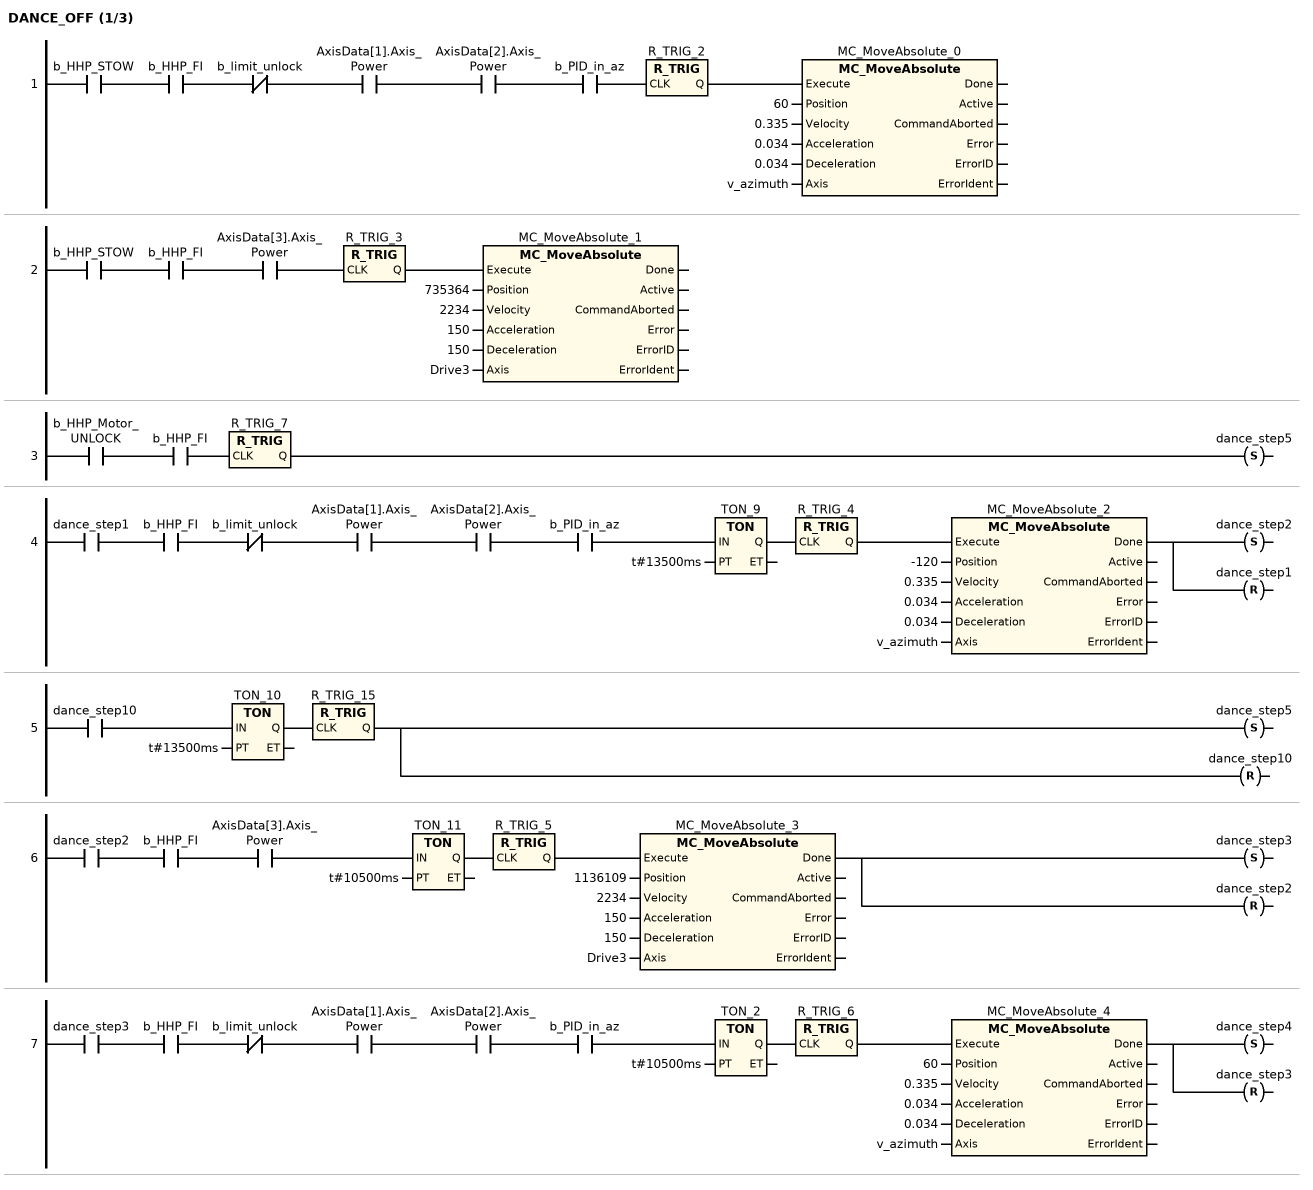
// NETWORK 1
R_TRIG_2(CLK := b_HHP_STOW AND b_HHP_FI AND NOT b_limit_unlock AND AxisData[1].Axis_Power AND AxisData[2].Axis_Power AND b_PID_in_az); // R_TRIG
MC_MoveAbsolute_0(
    Execute := R_TRIG_2.Q,
    Position := 60,
    Velocity := 0.335,
    Acceleration := 0.034,
    Deceleration := 0.034,
    Axis := v_azimuth); // MC_MoveAbsolute

// NETWORK 2
R_TRIG_3(CLK := b_HHP_STOW AND b_HHP_FI AND AxisData[3].Axis_Power); // R_TRIG
MC_MoveAbsolute_1(
    Execute := R_TRIG_3.Q,
    Position := 735364,
    Velocity := 2234,
    Acceleration := 150,
    Deceleration := 150,
    Axis := Drive3); // MC_MoveAbsolute

// NETWORK 3
R_TRIG_7(CLK := b_HHP_Motor_UNLOCK AND b_HHP_FI); // R_TRIG
dance_step5 S= R_TRIG_7.Q;

// NETWORK 4
TON_9(IN := dance_step1 AND b_HHP_FI AND NOT b_limit_unlock AND AxisData[1].Axis_Power AND AxisData[2].Axis_Power AND b_PID_in_az, PT := t#13500ms); // TON
R_TRIG_4(CLK := TON_9.Q); // R_TRIG
MC_MoveAbsolute_2(
    Execute := R_TRIG_4.Q,
    Position := -120,
    Velocity := 0.335,
    Acceleration := 0.034,
    Deceleration := 0.034,
    Axis := v_azimuth); // MC_MoveAbsolute
dance_step2 S= MC_MoveAbsolute_2.Done;
dance_step1 R= MC_MoveAbsolute_2.Done;

// NETWORK 5
TON_10(IN := dance_step10, PT := t#13500ms); // TON
R_TRIG_15(CLK := TON_10.Q); // R_TRIG
dance_step5 S= R_TRIG_15.Q;
dance_step10 R= R_TRIG_15.Q;

// NETWORK 6
TON_11(IN := dance_step2 AND b_HHP_FI AND AxisData[3].Axis_Power, PT := t#10500ms); // TON
R_TRIG_5(CLK := TON_11.Q); // R_TRIG
MC_MoveAbsolute_3(
    Execute := R_TRIG_5.Q,
    Position := 1136109,
    Velocity := 2234,
    Acceleration := 150,
    Deceleration := 150,
    Axis := Drive3); // MC_MoveAbsolute
dance_step3 S= MC_MoveAbsolute_3.Done;
dance_step2 R= MC_MoveAbsolute_3.Done;

// NETWORK 7
TON_2(IN := dance_step3 AND b_HHP_FI AND NOT b_limit_unlock AND AxisData[1].Axis_Power AND AxisData[2].Axis_Power AND b_PID_in_az, PT := t#10500ms); // TON
R_TRIG_6(CLK := TON_2.Q); // R_TRIG
MC_MoveAbsolute_4(
    Execute := R_TRIG_6.Q,
    Position := 60,
    Velocity := 0.335,
    Acceleration := 0.034,
    Deceleration := 0.034,
    Axis := v_azimuth); // MC_MoveAbsolute
dance_step4 S= MC_MoveAbsolute_4.Done;
dance_step3 R= MC_MoveAbsolute_4.Done;

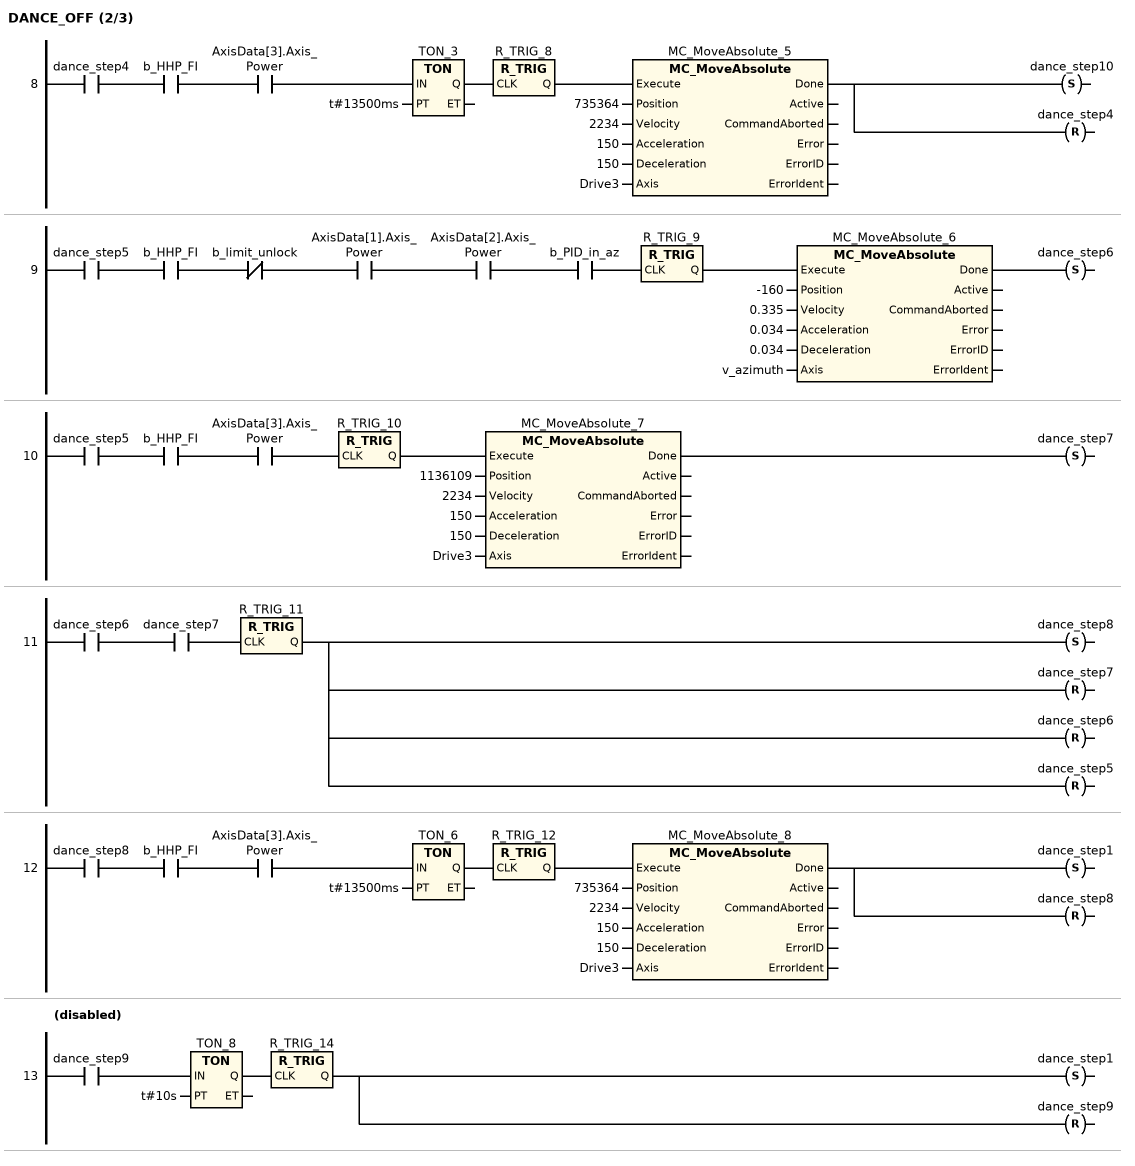
// NETWORK 8
TON_3(IN := dance_step4 AND b_HHP_FI AND AxisData[3].Axis_Power, PT := t#13500ms); // TON
R_TRIG_8(CLK := TON_3.Q); // R_TRIG
MC_MoveAbsolute_5(
    Execute := R_TRIG_8.Q,
    Position := 735364,
    Velocity := 2234,
    Acceleration := 150,
    Deceleration := 150,
    Axis := Drive3); // MC_MoveAbsolute
dance_step10 S= MC_MoveAbsolute_5.Done;
dance_step4 R= MC_MoveAbsolute_5.Done;

// NETWORK 9
R_TRIG_9(CLK := dance_step5 AND b_HHP_FI AND NOT b_limit_unlock AND AxisData[1].Axis_Power AND AxisData[2].Axis_Power AND b_PID_in_az); // R_TRIG
MC_MoveAbsolute_6(
    Execute := R_TRIG_9.Q,
    Position := -160,
    Velocity := 0.335,
    Acceleration := 0.034,
    Deceleration := 0.034,
    Axis := v_azimuth); // MC_MoveAbsolute
dance_step6 S= MC_MoveAbsolute_6.Done;

// NETWORK 10
R_TRIG_10(CLK := dance_step5 AND b_HHP_FI AND AxisData[3].Axis_Power); // R_TRIG
MC_MoveAbsolute_7(
    Execute := R_TRIG_10.Q,
    Position := 1136109,
    Velocity := 2234,
    Acceleration := 150,
    Deceleration := 150,
    Axis := Drive3); // MC_MoveAbsolute
dance_step7 S= MC_MoveAbsolute_7.Done;

// NETWORK 11
R_TRIG_11(CLK := dance_step6 AND dance_step7); // R_TRIG
dance_step8 S= R_TRIG_11.Q;
dance_step7 R= R_TRIG_11.Q;
dance_step6 R= R_TRIG_11.Q;
dance_step5 R= R_TRIG_11.Q;

// NETWORK 12
TON_6(IN := dance_step8 AND b_HHP_FI AND AxisData[3].Axis_Power, PT := t#13500ms); // TON
R_TRIG_12(CLK := TON_6.Q); // R_TRIG
MC_MoveAbsolute_8(
    Execute := R_TRIG_12.Q,
    Position := 735364,
    Velocity := 2234,
    Acceleration := 150,
    Deceleration := 150,
    Axis := Drive3); // MC_MoveAbsolute
dance_step1 S= MC_MoveAbsolute_8.Done;
dance_step8 R= MC_MoveAbsolute_8.Done;

// NETWORK 13 (disabled)
// TON_8(IN := dance_step9, PT := t#10s); // TON
// R_TRIG_14(CLK := TON_8.Q); // R_TRIG
// dance_step1 S= R_TRIG_14.Q;
// dance_step9 R= R_TRIG_14.Q;

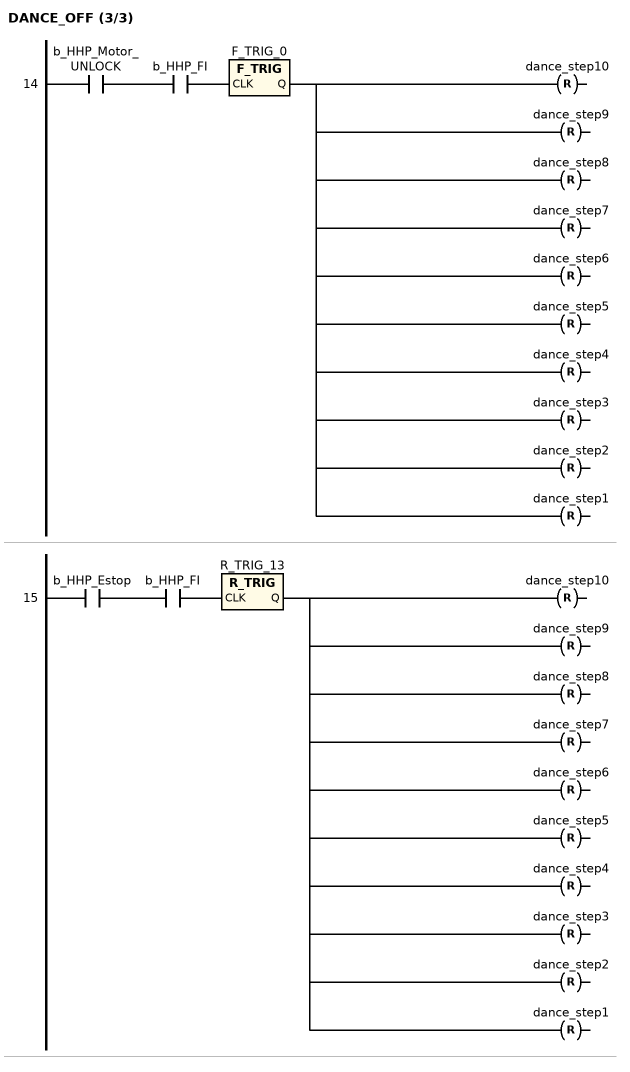
// NETWORK 14
F_TRIG_0(CLK := b_HHP_Motor_UNLOCK AND b_HHP_FI); // F_TRIG
dance_step10 R= F_TRIG_0.Q;
dance_step9 R= F_TRIG_0.Q;
dance_step8 R= F_TRIG_0.Q;
dance_step7 R= F_TRIG_0.Q;
dance_step6 R= F_TRIG_0.Q;
dance_step5 R= F_TRIG_0.Q;
dance_step4 R= F_TRIG_0.Q;
dance_step3 R= F_TRIG_0.Q;
dance_step2 R= F_TRIG_0.Q;
dance_step1 R= F_TRIG_0.Q;

// NETWORK 15
R_TRIG_13(CLK := b_HHP_Estop AND b_HHP_FI); // R_TRIG
dance_step10 R= R_TRIG_13.Q;
dance_step9 R= R_TRIG_13.Q;
dance_step8 R= R_TRIG_13.Q;
dance_step7 R= R_TRIG_13.Q;
dance_step6 R= R_TRIG_13.Q;
dance_step5 R= R_TRIG_13.Q;
dance_step4 R= R_TRIG_13.Q;
dance_step3 R= R_TRIG_13.Q;
dance_step2 R= R_TRIG_13.Q;
dance_step1 R= R_TRIG_13.Q;

END_PROGRAM

// IndraMotionMlc1/Application/POUs/Motion/P_Read_Parameters
(* The program is modified from the program that was built for GSTAT and KSTAT,according to ICD*)
PROGRAM P_Read_Parameters
VAR

(*The function block BLINK generates a pulsating signal.The input consists of ENABLE of the type BOOL, as well as TIMELOW and TIMEHIGH of the type TIME.*)
	fb_blink_diagnos_1: BLINK;
	fb_blink_diagnos_2: BLINK;
	fb_blink_diagnos_3: BLINK;
	fb_blink_diagnos_4: BLINK;
	fb_blink_diagnos_5: BLINK;
	fb_blink_diagnos_6: BLINK;
	fb_blink_diagnos_MLC: BLINK;
(*With the function block "MB_ReadParameter" it is possible to read the current value of a parameter. The return value is DINT*)
	fb_read_brake_1: MB_ReadParameter;
	fb_read_brake_2: MB_ReadParameter;
	fb_read_brake_3: MB_ReadParameter;
	fb_read_brake_4: MB_ReadParameter;
	fb_read_brake_5: MB_ReadParameter;
	fb_read_brake_6: MB_ReadParameter;
(*With the function block "MB_ReadStringParameter" it is possible to read a parameter the operating data of which has the ASCII format (string).*)
	fb_diagnose_1: MB_ReadStringParameter;
	fb_diagnose_2: MB_ReadStringParameter;
	fb_diagnose_3: MB_ReadStringParameter;
	fb_diagnose_4: MB_ReadStringParameter;
	fb_diagnose_5: MB_ReadStringParameter;
	fb_diagnose_6: MB_ReadStringParameter;
	fb_diagnose_MLC: MB_ReadStringParameter;
(*With the function block "MB_ReadRealParameter" it is possible to read the current value of a parameter. The return value is REAL. *)
	FB_readcur1: MB_ReadRealParameter;
	FB_readcur2: MB_ReadRealParameter;
	FB_readcur3: MB_ReadRealParameter;
	FB_readcur4: MB_ReadRealParameter;
	FB_readcur5: MB_ReadRealParameter;
	FB_readcur6: MB_ReadRealParameter;
	fb_temp_1: MB_ReadRealParameter;
	fb_temp_2: MB_ReadRealParameter;
	fb_temp_3: MB_ReadRealParameter;
	fb_temp_4: MB_ReadRealParameter;
	fb_temp_5: MB_ReadRealParameter;
	fb_temp_6: MB_ReadRealParameter;
	fb_read_s189_1: MB_ReadRealParameter;
	fb_read_s189_3: MB_ReadRealParameter;
	fb_read_s189_5: MB_ReadRealParameter;
	FB_readtor1: MB_ReadRealParameter;
	FB_readtor2: MB_ReadRealParameter;
	FB_readtor3: MB_ReadRealParameter;
	FB_readtor4: MB_ReadRealParameter;
	FB_readtor5: MB_ReadRealParameter;
	FB_readtor6: MB_ReadRealParameter;
	FB_temp_1_a: MB_ReadRealParameter;
	FB_temp_2_a: MB_ReadRealParameter;
	FB_temp_3_a: MB_ReadRealParameter;
	FB_temp_4_a: MB_ReadRealParameter;
	FB_temp_5_a: MB_ReadRealParameter;
	FB_temp_6_a: MB_ReadRealParameter;
(*FP_P_0_0539,Holding brake status word *)
	dw_brake_1: DWORD;
	dw_brake_2: DWORD;
	dw_brake_3: DWORD;
	dw_brake_4: DWORD;
	dw_brake_5: DWORD;
	dw_brake_6: DWORD;
(*FP_P_0_0007,Display text of diagnostic message*)
	str_diagnose_MLC: STRING;
	str_diagnose_1: STRING;
	str_diagnose_2: STRING;
	str_diagnose_3: STRING;
	str_diagnose_4: STRING;
	str_diagnose_5: STRING;
	str_diagnose_6: STRING;

(*FP_S_0_0384,Amplifier temperature*)
	r_temp_amp1: REAL;
	r_temp_amp2: REAL;
	r_temp_amp3: REAL;
	r_temp_amp4: REAL;
	r_temp_amp5: REAL;
	r_temp_amp6: REAL;


(*<<<<<<<<<<<<<<<<<<<<<<<<<<<<<<<<<<<<<<<add MLC temperature and operation hour(20100708)>>>>>>>>>>>>>>>>>>>>>>>>>>>>>>>>>>>>>*)
	fb_temp_MLC: MB_ReadRealParameter;
	r_temp_MLC: REAL;(*FP_c_0_0070,Control unit temperature*)
	fb_read_system_status: MB_ReadParameter;
	dw_system_status: DWORD;(*FP_C_0_0023,MC system status,used for temperature warning*)
	fb_read_operation_hour: MB_ReadParameter;

(*the limit for judging whether azimuth following error is too big*)
	r_limit_track_az: REAL;
(*test for limit check*)
	fb_software_limit_1: MB_ReadParameter;
	fb_software_limit_5: MB_ReadParameter;
	fb_software_limit_3: MB_ReadParameter;
	fb_hardware_limit_1: MB_ReadParameter;
	fb_hardware_limit_3: MB_ReadParameter;
	fb_hardware_limit_5: MB_ReadParameter;
	fb_ESTOP_1: MB_ReadParameter;
	fb_ESTOP_3: MB_ReadParameter;
	fb_ESTOP_5: MB_ReadParameter;
	i_software_limit_1: DINT;
	i_software_limit_3: DINT;
	i_software_limit_5: DINT;
	i_hardware_limit_1: DINT;
	i_hardware_limit_3: DINT;
	i_hardware_limit_5: DINT;
	i_ESTOP_1: DINT;
	i_ESTOP_3: DINT;
	i_ESTOP_5: DINT;


	b_azimuth_limit: BOOL;
	b_elevation_limit: BOOL;
	b_FeedIndexer_limit: BOOL;
	fb_readpar_speed_1: MB_ReadRealParameter;
	fb_readpar_speed_3: MB_ReadRealParameter;
	fb_readpar_speed_5: MB_ReadRealParameter;
	
	str_concat: ARRAY[1..40] OF STRING(1500);(*数组及其类型的定义*)	
	Counter: INT;
	FB_readmotorencoder1: MB_ReadRealParameter;
	FB_readmotorencoder2: MB_ReadRealParameter;
	FB_readmotorencoder3: MB_ReadRealParameter;
	FB_readmotorencoder4: MB_ReadRealParameter;
	FB_readmotorencoder5: MB_ReadRealParameter;
	FB_readmotorencoder6: MB_ReadRealParameter;
	r_motorencoder_6: REAL;
	r_motorencoder_5: REAL;
	r_motorencoder_4: REAL;
	r_motorencoder_3: REAL;
	r_motorencoder_2: REAL;
	r_motorencoder_1: REAL;
	
	(*the status word for GSTAT*)
	
	status_1:DWORD;
	status_2:DWORD;
	status_3:DWORD;
	status_4:DWORD;
	status_5:DWORD;
	status_6:DWORD;
	fb_diagnose_111: MB_ReadParameter;
	str_diagnose_11: DWORD;
	fb_blink_diagnos_11: BLINK;
	fb_diagnose_11: MB_ReadrealParameter;
	str_diagnose_111: REAL;
	fb_readpar_speed_2: MB_ReadRealParameter;
	fb_readpar_speed_4: MB_ReadRealParameter;
	fb_readpar_speed_6: MB_ReadRealParameter;
	
	ReadAxisPshape: ARRAY[1..5] OF MB_ReadlrealParameter;
	ReadAxisVact: ARRAY[1..5] OF MB_ReadlrealParameter;
	ReadAxisVshape: ARRAY[1..5] OF MB_ReadlrealParameter;

	conut_i: INT;
	b_PID_in_FI: BOOL;
	b_limit_cw_FI: BOOL;
	b_limit_ccw_FI: BOOL;
	b_limit_final_FI: BOOL;
	fb_readpar_pos_cmd_1: MB_ReadRealParameter;
END_VAR

P_Read_Parameters.A_Read_Parameter();

status_code1:=LEFT(str_diagnose_1,5);
status_code2:=LEFT(str_diagnose_2,5);
status_code3:=LEFT(str_diagnose_3,5);
status_code4:=LEFT(str_diagnose_4,5);
status_code5:=LEFT(str_diagnose_5,5);
status_code6:=LEFT(str_diagnose_6,5);

FOR  conut_i:=1 TO 5 BY 1 DO
ReadAxisPshape[conut_i](
	Enable:=axisdata[1].Axis_Inbb , 
	Done=> , 
	Active=> , 
	Error=> , 
	ErrorID=> , 
	ErrorIdent=> , 
	ParameterNumber:=FP_P_0_0434 , 
	Value=>P_shape_value[conut_i] , 
	Axis:=AxRef[conut_i] );
	
ReadAxisVshape[conut_i](
	Enable:=axisdata[1].Axis_Inbb , 
	Done=> , 
	Active=> , 
	Error=> , 
	ErrorID=> , 
	ErrorIdent=> , 
	ParameterNumber:=FP_P_0_0434 , 
	Value=>V_shape_value[conut_i] , 
	Axis:=AxRef[conut_i] );
	
ReadAxisVact[conut_i](
	Enable:=axisdata[1].Axis_Inbb , 
	Done=> , 
	Active=> , 
	Error=> , 
	ErrorID=> , 
	ErrorIdent=> , 
	ParameterNumber:=FP_S_0_0040 , 
	Value=>V_act_value[conut_i] , 
	Axis:=AxRef[conut_i] );
END_FOR
(*
(*<<<<<<<<<<<<<<<<<<<<<<<<<<<<<master_status>>>>>>>>>>>>>>>>>>>>>>>>>>>>>>>>>>>>>>>>>>>>>>>>>>>>>>>*)
master_status.0:=axisdata[1].Axis_InAb;
IF b_remote_on=TRUE THEN
	master_status.1:=0;
ELSE
	master_status.1:=1;
END_IF
IF b_DSdoor_Estop  THEN
	master_status.2:=1;
ELSE
	master_status.2:=0;
END_IF

IF ABS(axisdata[3].rActualPosition_i-90)<0.02 THEN
	master_status.3:=1;
ELSE
	master_status.3:=0;
END_IF
	master_status.4:=(axisdata[1].Axis_Error OR axisdata[2].Axis_Error OR axisdata[3].Axis_Error OR axisdata[4].Axis_Error OR axisdata[5].Axis_Error OR axisdata[6].Axis_Error);
	master_status.5:=b_stow_pin_limit_unlock;
	master_status.6:=b_stow_pin_limit_lock;
	
IF i_num_stack_left>9500 THEN
		master_status.7:=0;
	ELSE IF i_num_stack_left<1500 THEN
		master_status.7:=1;	
	END_IF
		
END_IF

IF b_remote_on_run AND b_track_on THEN
	master_status.9:=0;
	master_status.8:=1;
ELSIF b_remote_on_run AND b_Track_Pause = TRUE THEN
	master_status.9:=1;
	master_status.8:=0;
ELSIF b_remote_on_run AND b_Track_Pause = FALSE  AND b_track_on = FALSE THEN
	master_status.9:=0;
	master_status.8:=0;
ELSE
 	master_status.9:=1;
	master_status.8:=1;
END_IF

IF 	b_encoder_ok_az	AND b_encoder_ok_FI THEN
	master_status.10:=1;
	master_status.11:=1;
ELSIF b_encoder_ok_az =FALSE AND b_encoder_ok_FI THEN
	master_status.10:=0;
	master_status.11:=1;
ELSIF b_encoder_ok_az  AND b_encoder_ok_FI=FALSE THEN
	master_status.10:=1;
	master_status.11:=0;
ELSE
	master_status.10:=0;
	master_status.11:=0;		
END_IF

IF b_remote_on_run THEN
	master_status.12:=1;
ELSE
	master_status.12:=0;
END_IF
	
IF b_remote_on_run THEN
	master_status.12:=1;
ELSE
	master_status.12:=0;
END_IF

IF b_permit_new_file THEN
	master_status.13:=1;
ELSE
	master_status.13:=0;
END_IF

(*<<<<<<<<<<<<<<<<<<<<<<<<<<<<<status_1>>>>>>>>>>>>>>>>>>>>>>>>>>>>>>>>>>>>>>>>>>>>>>>>>>>>>>>*)
status_1.0:=axisdata[1].Axis_InAb;
status_1.1:=b_PID_in_az;
status_1.2:=dw_brake_1.0;
status_1.3:=b_limit_cw_az;
status_1.4:=b_limit_ccw_az;
status_1.5:=(b_limit_final_cw_az OR b_limit_final_ccw_az);
status_1.6:=axisdata[1].Axis_Error;

(*<<<<<<<<<<<<<<<<<<<<<<<<<<<<<status_2>>>>>>>>>>>>>>>>>>>>>>>>>>>>>>>>>>>>>>>>>>>>>>>>>>>>>>>*)
status_2.0:=axisdata[2].Axis_InAb;
status_2.1:=b_PID_in_az;
status_2.2:=dw_brake_2.0;
status_2.3:=b_limit_cw_az;
status_2.4:=b_limit_ccw_az;
status_2.5:=(b_limit_final_cw_az OR b_limit_final_ccw_az);
status_2.6:=axisdata[2].Axis_Error;

(*<<<<<<<<<<<<<<<<<<<<<<<<<<<<<status_3>>>>>>>>>>>>>>>>>>>>>>>>>>>>>>>>>>>>>>>>>>>>>>>>>>>>>>>*)
status_3.0:=axisdata[3].Axis_InAb;
status_3.1:=b_PID_in_el;
status_3.2:=dw_brake_3.0;
status_3.3:=b_limit_cw_el;
status_3.4:=b_limit_ccw_el;
status_3.5:=(b_limit_final_cw_el OR b_limit_final_ccw_el) ;
status_3.6:=axisdata[3].Axis_Error;

(*<<<<<<<<<<<<<<<<<<<<<<<<<<<<<status_4>>>>>>>>>>>>>>>>>>>>>>>>>>>>>>>>>>>>>>>>>>>>>>>>>>>>>>>*)
status_4.0:=axisdata[4].Axis_InAb;
status_4.1:=b_PID_in_el;
status_4.2:=dw_brake_4.0;
status_4.3:=b_limit_cw_el;
status_4.4:=b_limit_ccw_el;
status_4.5:=(b_limit_final_cw_el OR b_limit_final_ccw_el); 
status_4.6:=axisdata[4].Axis_Error;

(*<<<<<<<<<<<<<<<<<<<<<<<<<<<<<status_5>>>>>>>>>>>>>>>>>>>>>>>>>>>>>>>>>>>>>>>>>>>>>>>>>>>>>>>*)
status_5.0:=axisdata[5].Axis_InAb;
status_5.1:=b_PID_in_FI;
status_5.2:=dw_brake_5.0;
status_5.3:=b_limit_cw_FI;
status_5.4:=b_limit_ccw_FI;
status_5.5:=b_limit_final_FI;
status_5.6:=axisdata[5].Axis_Error;

(*<<<<<<<<<<<<<<<<<<<<<<<<<<<<<status_6>>>>>>>>>>>>>>>>>>>>>>>>>>>>>>>>>>>>>>>>>>>>>>>>>>>>>>>*)
status_6.0:=axisdata[6].Axis_InAb;
status_6.1:=b_PID_in_FI;
status_6.2:=dw_brake_6.0;
status_6.3:=b_limit_cw_FI;
status_6.4:=b_limit_ccw_FI;
status_6.5:=b_limit_final_FI;
status_6.6:=axisdata[6].Axis_Error;


(*
(*<<<<<<<<<<<<<<<<<<<<<<<<<<<<<status_2>>>>>>>>>>>>>>>>>>>>>>>>>>>>>>>>>>>>>>>>>>>>>>>>>>>>>>>*)
status_2.0:=NOT(axisdata[2].Axis_InAb);
status_2.1:=axisdata[2].Axis_Error;
status_2.2:=NOT(dw_brake_2.0);
IF r_temp_motor2>120 THEN
status_2.3:=1;
b_power_Az:=FALSE;
b_enable_az_1:=FALSE;
b_enable_az_2:=FALSE;
ELSE
status_2.3:=0;
END_IF
IF r_current_2>5 THEN
status_2.4:=1;
ELSE
status_2.4:=0;
END_IF
(*<<<<<<<<<<<<<<<<<<<<<<<<<<<<<status_3>>>>>>>>>>>>>>>>>>>>>>>>>>>>>>>>>>>>>>>>>>>>>>>>>>>>>>>*)
status_3.0:=NOT(axisdata[3].Axis_InAb);
status_3.1:=axisdata[3].Axis_Error;
status_3.2:=NOT(dw_brake_3.0);
IF r_temp_motor3>120 THEN
status_3.3:=1;
b_power_El:=FALSE;
b_enable_el_3:=FALSE;
b_enable_el_4:=FALSE;
ELSE
status_3.3:=0;
END_IF
IF r_current_3>5 THEN
status_3.4:=1;
ELSE
status_3.4:=0;
END_IF
status_3.8:=NOT(b_PID_in_el);

IF (b_scc_goto=TRUE AND (b_goto_Az_done=FALSE OR b_goto_El_done=FALSE OR b_goto_FI_done=FALSE)) OR (b_track_on=TRUE AND i_num_stack_left<>0) THEN
status_3.9:=1;
END_IF;
IF (b_goto_Az_done=TRUE AND b_goto_El_done=TRUE AND b_goto_FI_done=TRUE) OR i_num_stack_left=0 THEN
status_3.9:=0;
END_IF;

status_3.10:=NOT(b_track_on);
IF ABS(r_track_error[2])<0.0034 THEN
	status_3.11:=0;
ELSE
	status_3.11:=1;
END_IF
status_3.12:=axisdata[3].Axis_Error;
IF ABS(r_following_3)>0.5 THEN
status_3.13:=1;
ELSE
status_3.13:=0;
END_IF
IF r_pos_el<14.6 THEN
	status_3.14:=1;
ELSE
	status_3.14:=0;
END_IF
IF r_pos_el>90.15 THEN
	status_3.15:=1;
ELSE
	status_3.15:=0;
END_IF
status_3.16:=b_limit_ccw_el;
status_3.17:=b_limit_cw_el;
status_3.18:=b_limit_final_el;
status_3.19:=b_track_overspeed_el;
(*<<<<<<<<<<<<<<<<<<<<<<<<<<<<<status_4>>>>>>>>>>>>>>>>>>>>>>>>>>>>>>>>>>>>>>>>>>>>>>>>>>>>>>>*)
status_4.0:=NOT(axisdata[4].Axis_InAb);
status_4.1:=axisdata[4].Axis_Error;
status_4.2:=NOT(dw_brake_4.0);
IF r_temp_motor4>120 THEN
status_4.3:=1;
b_power_El:=FALSE;
b_enable_el_3:=FALSE;
b_enable_el_4:=FALSE;
ELSE
status_4.3:=0;
END_IF
IF r_current_4>5 THEN
status_4.4:=1;
ELSE
status_4.4:=0;
END_IF
(*<<<<<<<<<<<<<<<<<<<<<<<<<<<<<status_5>>>>>>>>>>>>>>>>>>>>>>>>>>>>>>>>>>>>>>>>>>>>>>>>>>>>>>>*)
status_5.0:=NOT(axisdata[5].Axis_InAb);
status_5.1:=axisdata[5].Axis_Error;
status_5.2:=NOT(dw_brake_5.0);
IF r_temp_motor5>120 THEN
status_5.3:=1;
b_power_FI:=FALSE;
b_enable_FI_5:=FALSE;
ELSE
status_5.3:=0;
END_IF
IF r_current_5>5 THEN
status_5.4:=1;
ELSE
status_5.4:=0;
END_IF

status_5.8:=NOT(b_gearinpos_5_done);

IF (b_scc_goto=TRUE AND (b_goto_Az_done=FALSE OR b_goto_El_done=FALSE OR b_goto_FI_done=FALSE)) OR (b_track_on=TRUE AND i_num_stack_left<>0) THEN
status_5.9:=1;
END_IF;
IF (b_goto_Az_done=TRUE AND b_goto_El_done=TRUE AND b_goto_FI_done=TRUE) OR i_num_stack_left=0 THEN
status_5.9:=0;
END_IF;

status_5.10:=NOT(b_track_on);
IF ABS(r_track_error[3])<0.0034 THEN
	status_5.11:=0;
ELSE
	status_5.11:=1;
END_IF
status_5.12:=axisdata[5].Axis_Error;
IF ABS(r_following_5)>0.5 THEN
status_5.13:=1;
ELSE
status_5.13:=0;
END_IF

IF r_pos_FI<-89 THEN
	status_5.14:=1;
ELSE
	status_5.14:=0;
END_IF

IF r_pos_FI>89 THEN
	status_5.15:=1;
ELSE
	status_5.15:=0;
END_IF
status_5.16:=b_limit_ccw_FI;
status_5.17:=b_limit_cw_FI;
status_5.18:=b_limit_final_FI;
status_5.19:=b_track_overspeed_FI;
*)

(*<<<<<<<<<<<<<<<<<<<<<<<<<<<<<concatenate STR_GSTAT>>>>>>>>>>>>>>>>>>>>>>>>>>>>>>>>>>>>>>>>>>>>>>>>>>>>>>>*)
(*
str_concat[1]:=CONCAT(' ',DWORD_TO_STRING(status_1));
str_concat[2]:=CONCAT(' ',LREAL_TO_STRING(F_reduce_to_1_bit(LREAL_TO_STRING(r_current_1))));
str_concat[3]:=CONCAT(' ',LREAL_TO_STRING(r_temp_motor1));
str_concat[4]:=CONCAT(' ',LREAL_TO_STRING(i_speed_1));
str_concat[5]:=CONCAT(' ',LREAL_TO_STRING(F_reduce_to_1_bit(LREAL_TO_STRING(r_motorencoder_1))));


str_concat[6]:=CONCAT(' ',DWORD_TO_STRING(status_2));
str_concat[7]:=CONCAT(' ',LREAL_TO_STRING(F_reduce_to_1_bit(LREAL_TO_STRING(r_current_2))));
str_concat[8]:=CONCAT(' ',LREAL_TO_STRING(r_temp_motor2));
str_concat[9]:=CONCAT(' ',LREAL_TO_STRING(i_speed_2));
str_concat[10]:=CONCAT(' ',LREAL_TO_STRING(F_reduce_to_1_bit(LREAL_TO_STRING(r_motorencoder_2))));

str_concat[11]:=CONCAT(' ',DWORD_TO_STRING(status_3));
str_concat[12]:=CONCAT(' ',LREAL_TO_STRING(F_reduce_to_1_bit(LREAL_TO_STRING(r_current_3))));
str_concat[13]:=CONCAT(' ',LREAL_TO_STRING(r_temp_motor3));
str_concat[14]:=CONCAT(' ',LREAL_TO_STRING(i_speed_3));
str_concat[15]:=CONCAT(' ',LREAL_TO_STRING(F_reduce_to_1_bit(LREAL_TO_STRING(r_motorencoder_3))));

str_concat[16]:=CONCAT(' ',DWORD_TO_STRING(status_4));
str_concat[17]:=CONCAT(' ',LREAL_TO_STRING(F_reduce_to_1_bit(LREAL_TO_STRING(r_current_4))));
str_concat[18]:=CONCAT(' ',LREAL_TO_STRING(r_temp_motor4));
str_concat[19]:=CONCAT(' ',LREAL_TO_STRING(i_speed_4));
str_concat[20]:=CONCAT(' ',LREAL_TO_STRING(F_reduce_to_1_bit(LREAL_TO_STRING(r_motorencoder_4))));

str_concat[21]:=CONCAT(' ',DWORD_TO_STRING(status_5));
str_concat[22]:=CONCAT(' ',LREAL_TO_STRING(F_reduce_to_1_bit(LREAL_TO_STRING(r_current_5))));
str_concat[23]:=CONCAT(' ',LREAL_TO_STRING(r_temp_motor5));
str_concat[24]:=CONCAT(' ',LREAL_TO_STRING(i_speed_5));
str_concat[25]:=CONCAT(' ',LREAL_TO_STRING(F_reduce_to_1_bit(LREAL_TO_STRING(r_motorencoder_5))));

str_concat[26]:=CONCAT(' ',DWORD_TO_STRING(status_6));
str_concat[27]:=CONCAT(' ',LREAL_TO_STRING(F_reduce_to_1_bit(LREAL_TO_STRING(r_current_6))));
str_concat[28]:=CONCAT(' ',LREAL_TO_STRING(r_temp_motor6));
str_concat[29]:=CONCAT(' ',LREAL_TO_STRING(i_speed_6));
str_concat[30]:=CONCAT(' ',LREAL_TO_STRING(F_reduce_to_1_bit(LREAL_TO_STRING(r_motorencoder_6))));

str_concat[31]:=CONCAT(' ',last_command);
str_concat[32]:=CONCAT(' ',INT_TO_STRING(i_receive_cmd));
str_concat[33]:=CONCAT(' ',INT_TO_STRING(i_excute_cmd));
(*
str_concat[31]:=CONCAT(' ',REAL_TO_STRING(F_reduce_to_4_bit(REAL_TO_STRING(r_test1))));
str_concat[32]:=CONCAT(' ',REAL_TO_STRING(F_reduce_to_4_bit(REAL_TO_STRING(r_test2))));
str_concat[33]:=CONCAT(' ',REAL_TO_STRING(F_reduce_to_4_bit(REAL_TO_STRING(r_test3))));
*)

STR_GSTAT_M:='';(*for语句格式*)
				FOR Counter:=1 TO 33 BY 1 DO
					STR_GSTAT_M:=CONCAT(STR_GSTAT_M,str_concat[Counter]);
				END_FOR;



(*
STR_GSTAT:=CONCAT(STR_GSTAT,CONCAT(' ',DWORD_TO_STRING(status_1)));
STR_GSTAT:=CONCAT(STR_GSTAT,CONCAT(' ',REAL_TO_STRING(r_current_1)));
STR_GSTAT:=CONCAT(STR_GSTAT,CONCAT(' ',REAL_TO_STRING(r_temp_motor1)));
STR_GSTAT:=CONCAT(STR_GSTAT,CONCAT(' ',REAL_TO_STRING(i_speed_1)));
*)


(*
STR_GSTAT:=CONCAT(STR_GSTAT,CONCAT(' ',DWORD_TO_STRING(status_2)));
STR_GSTAT:=CONCAT(STR_GSTAT,CONCAT(' ',REAL_TO_STRING(r_current_2)));
STR_GSTAT:=CONCAT(STR_GSTAT,CONCAT(' ',REAL_TO_STRING(r_temp_motor2)));
STR_GSTAT:=CONCAT(STR_GSTAT,CONCAT(' ',REAL_TO_STRING(i_speed_1)));

STR_GSTAT:=CONCAT(STR_GSTAT,CONCAT(' ',DWORD_TO_STRING(status_3)));
STR_GSTAT:=CONCAT(STR_GSTAT,CONCAT(' ',REAL_TO_STRING(r_current_3)));
STR_GSTAT:=CONCAT(STR_GSTAT,CONCAT(' ',REAL_TO_STRING(r_temp_motor3)));
STR_GSTAT:=CONCAT(STR_GSTAT,CONCAT(' ',REAL_TO_STRING(i_speed_3)));

STR_GSTAT:=CONCAT(STR_GSTAT,CONCAT(' ',DWORD_TO_STRING(status_4)));
STR_GSTAT:=CONCAT(STR_GSTAT,CONCAT(' ',REAL_TO_STRING(r_current_4)));
STR_GSTAT:=CONCAT(STR_GSTAT,CONCAT(' ',REAL_TO_STRING(r_temp_motor4)));
STR_GSTAT:=CONCAT(STR_GSTAT,CONCAT(' ',REAL_TO_STRING(i_speed_3)));

STR_GSTAT:=CONCAT(STR_GSTAT,CONCAT(' ',DWORD_TO_STRING(status_5)));
STR_GSTAT:=CONCAT(STR_GSTAT,CONCAT(' ',REAL_TO_STRING(r_current_5)));
STR_GSTAT:=CONCAT(STR_GSTAT,CONCAT(' ',REAL_TO_STRING(r_temp_motor5)));
STR_GSTAT:=CONCAT(STR_GSTAT,CONCAT(' ',REAL_TO_STRING(i_speed_5)));

STR_GSTAT:=CONCAT(STR_GSTAT,CONCAT(' ',DWORD_TO_STRING(status_6)));
STR_GSTAT:=CONCAT(STR_GSTAT,CONCAT(' ',REAL_TO_STRING(r_current_6)));
STR_GSTAT:=CONCAT(STR_GSTAT,CONCAT(' ',REAL_TO_STRING(r_temp_motor6)));
STR_GSTAT:=CONCAT(STR_GSTAT,CONCAT(' ',REAL_TO_STRING(i_speed_5)));

STR_GSTAT:=CONCAT(STR_GSTAT,CONCAT(' ',INT_TO_STRING(i_num_stack_left)));
STR_GSTAT:=CONCAT(STR_GSTAT,CONCAT(' ',INT_TO_STRING(i_start)));
STR_GSTAT_M:=CONCAT(STR_GSTAT,CONCAT(' ',INT_TO_STRING(i_end)));

*)
(*
(*<<<<<<<<<<<<<<<<<<<<<<<<<<<<<concatenate STR_K2STAT>>>>>>>>>>>>>>>>>>>>>>>>>>>>>>>>>>>>>>>>>>>>>>>>>>>>>>>*)
STR_K2STAT:=CONCAT('OK - ',REAL_TO_STRING(r_operation_hour/100));
STR_K2STAT:=CONCAT(STR_K2STAT,CONCAT(' ',LREAL_TO_STRING(r_temp_motor1)));
STR_K2STAT:=CONCAT(STR_K2STAT,CONCAT(' ',LREAL_TO_STRING(r_temp_motor2)));
STR_K2STAT:=CONCAT(STR_K2STAT,CONCAT(' ',LREAL_TO_STRING(r_temp_motor3)));
STR_K2STAT:=CONCAT(STR_K2STAT,CONCAT(' ',LREAL_TO_STRING(r_temp_motor4)));
STR_K2STAT:=CONCAT(STR_K2STAT,CONCAT(' ',LREAL_TO_STRING(r_temp_motor5)));
STR_K2STAT:=CONCAT(STR_K2STAT,CONCAT(' ',LREAL_TO_STRING(r_temp_amp1)));
STR_K2STAT:=CONCAT(STR_K2STAT,CONCAT(' ',LREAL_TO_STRING(r_temp_amp2)));
STR_K2STAT:=CONCAT(STR_K2STAT,CONCAT(' ',LREAL_TO_STRING(r_temp_amp3)));
STR_K2STAT:=CONCAT(STR_K2STAT,CONCAT(' ',LREAL_TO_STRING(r_temp_amp4)));
STR_K2STAT:=CONCAT(STR_K2STAT,CONCAT(' ',LREAL_TO_STRING(r_temp_amp5)));
STR_K2STAT_M:=CONCAT(STR_K2STAT,CONCAT(' ',LREAL_TO_STRING(r_temp_MLC)));
(*<<<<<<<<<<<<<<<<<<<<<<<<<<<<<concatenate STR_K4STAT>>>>>>>>>>>>>>>>>>>>>>>>>>>>>>>>>>>>>>>>>>>>>>>>>>>>>>>*)
STR_K4STAT:=CONCAT('OK - ',str_diagnose_MLC);
STR_K4STAT:=CONCAT(STR_K4STAT,CONCAT(' ',str_diagnose_1));
STR_K4STAT:=CONCAT(STR_K4STAT,CONCAT(' ',str_diagnose_2));
STR_K4STAT:=CONCAT(STR_K4STAT,CONCAT(' ',str_diagnose_3));
STR_K4STAT:=CONCAT(STR_K4STAT,CONCAT(' ',str_diagnose_4));
STR_K4STAT_M:=CONCAT(STR_K4STAT,CONCAT(' ',str_diagnose_5));

(*<<<<<<<<<<<<<<<<<<<<<<<<<<<<<concatenate STR_K5STAT>>>>>>>>>>>>>>>>>>>>>>>>>>>>>>>>>>>>>>>>>>>>>>>>>>>>>>>*)
IF i_software_limit_1=16 AND i_hardware_limit_1=3 AND i_ESTOP_1=5 THEN
	b_azimuth_limit:=TRUE;
ELSE
	b_azimuth_limit:=FALSE;
END_IF

IF i_software_limit_3=16 AND i_hardware_limit_3=3 AND i_ESTOP_3=5 THEN
	b_elevation_limit:=TRUE;
ELSE
	b_elevation_limit:=FALSE;
END_IF

IF i_software_limit_5=16 AND i_hardware_limit_5=3 AND i_ESTOP_5=5 THEN
	b_FeedIndexer_limit:=TRUE;
ELSE
	b_FeedIndexer_limit:=FALSE;
END_IF
IF b_azimuth_limit AND b_elevation_limit AND b_FeedIndexer_limit THEN
	STR_K5STAT_M:='All the axes are safe.';
ELSE
	STR_K5STAT_M:='';
	IF b_azimuth_limit=FALSE THEN
		STR_K5STAT_M:=CONCAT(STR_K5STAT_M,'Azimuth axis is unsafe. ');
	END_IF
	IF b_elevation_limit=FALSE THEN
		STR_K5STAT_M:=CONCAT(STR_K5STAT_M,'Elevation axis is unsafe. ');
	END_IF
	IF b_FeedIndexer_limit=FALSE THEN
		STR_K5STAT_M:=CONCAT(STR_K5STAT_M,'FeedIndexer axis is unsafe. ');
	END_IF
END_IF*)*) *)

ACTION A_Read_Parameter:
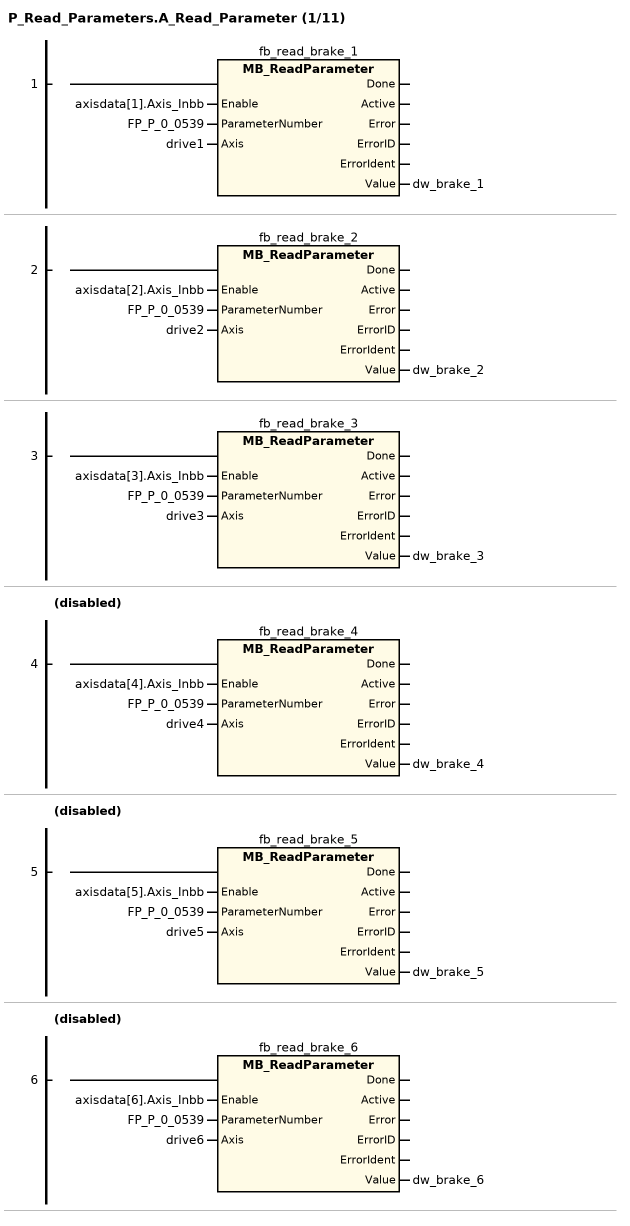
// NETWORK 1
//   fb_read_brake_1: With the function block "MB_ReadParameter" it is possible to read the current value of a parameter. The return value is DINT
//   axisdata[1].Axis_Inbb: A-0-0021.13 -RD- Axis is ready for power to the amplifier (bb)
//   FP_P_0_0539: Holding brake status word
//   drive1: Real axis "Drive1" with axis number 1
//   dw_brake_1: FP_P_0_0539,Holding brake status word
fb_read_brake_1(
    Enable := axisdata[1].Axis_Inbb,
    ParameterNumber := FP_P_0_0539,
    Axis := drive1,
    Value => dw_brake_1); // MB_ReadParameter

// NETWORK 2
//   axisdata[2].Axis_Inbb: A-0-0021.13 -RD- Axis is ready for power to the amplifier (bb)
//   FP_P_0_0539: Holding brake status word
//   drive2: Real axis "Drive2" with axis number 2
fb_read_brake_2(
    Enable := axisdata[2].Axis_Inbb,
    ParameterNumber := FP_P_0_0539,
    Axis := drive2,
    Value => dw_brake_2); // MB_ReadParameter

// NETWORK 3
//   axisdata[3].Axis_Inbb: A-0-0021.13 -RD- Axis is ready for power to the amplifier (bb)
//   FP_P_0_0539: Holding brake status word
//   drive3: Real axis "Drive3" with axis number 3
fb_read_brake_3(
    Enable := axisdata[3].Axis_Inbb,
    ParameterNumber := FP_P_0_0539,
    Axis := drive3,
    Value => dw_brake_3); // MB_ReadParameter

// NETWORK 4 (disabled)
//   axisdata[4].Axis_Inbb: A-0-0021.13 -RD- Axis is ready for power to the amplifier (bb)
//   FP_P_0_0539: Holding brake status word
//   drive4: Real axis "Drive4" with axis number 4
// fb_read_brake_4(
//     Enable := axisdata[4].Axis_Inbb,
//     ParameterNumber := FP_P_0_0539,
//     Axis := drive4,
//     Value => dw_brake_4); // MB_ReadParameter

// NETWORK 5 (disabled)
//   axisdata[5].Axis_Inbb: A-0-0021.13 -RD- Axis is ready for power to the amplifier (bb)
//   FP_P_0_0539: Holding brake status word
//   drive5: Real axis "Drive5" with axis number 5
// fb_read_brake_5(
//     Enable := axisdata[5].Axis_Inbb,
//     ParameterNumber := FP_P_0_0539,
//     Axis := drive5,
//     Value => dw_brake_5); // MB_ReadParameter

// NETWORK 6 (disabled)
//   axisdata[6].Axis_Inbb: A-0-0021.13 -RD- Axis is ready for power to the amplifier (bb)
//   FP_P_0_0539: Holding brake status word
//   drive6: Real axis "Drive6" with axis number 6
// fb_read_brake_6(
//     Enable := axisdata[6].Axis_Inbb,
//     ParameterNumber := FP_P_0_0539,
//     Axis := drive6,
//     Value => dw_brake_6); // MB_ReadParameter

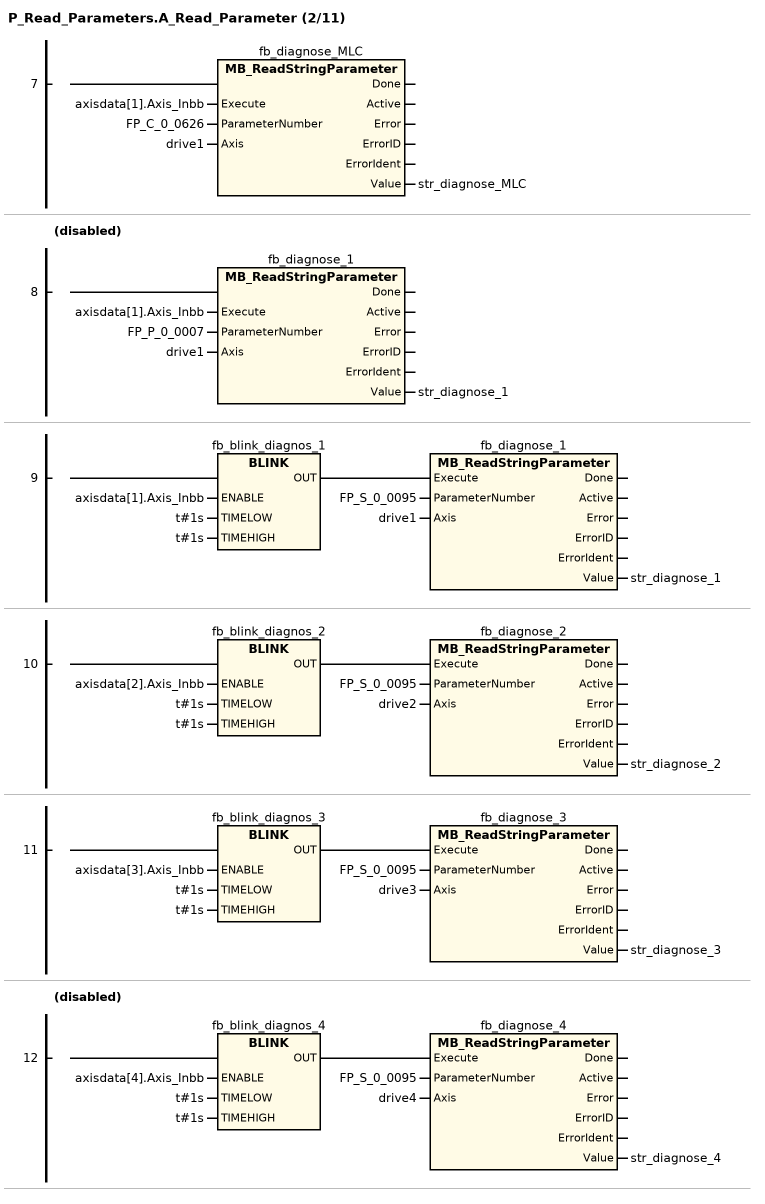
// NETWORK 7
//   axisdata[1].Axis_Inbb: A-0-0021.13 -RD- Axis is ready for power to the amplifier (bb)
//   FP_C_0_0626: Diagnostics
//   drive1: Real axis "Drive1" with axis number 1
//   str_diagnose_MLC: FP_P_0_0007,Display text of diagnostic message
fb_diagnose_MLC(
    Execute := axisdata[1].Axis_Inbb,
    ParameterNumber := FP_C_0_0626,
    Axis := drive1,
    Value => str_diagnose_MLC); // MB_ReadStringParameter

// NETWORK 8 (disabled)
//   fb_diagnose_1: With the function block "MB_ReadStringParameter" it is possible to read a parameter the operating data of which has the ASCII format (string).
//   axisdata[1].Axis_Inbb: A-0-0021.13 -RD- Axis is ready for power to the amplifier (bb)
//   FP_P_0_0007: Display text of diagnostic message
//   drive1: Real axis "Drive1" with axis number 1
// fb_diagnose_1(
//     Execute := axisdata[1].Axis_Inbb,
//     ParameterNumber := FP_P_0_0007,
//     Axis := drive1,
//     Value => str_diagnose_1); // MB_ReadStringParameter

// NETWORK 9
//   fb_diagnose_1: With the function block "MB_ReadStringParameter" it is possible to read a parameter the operating data of which has the ASCII format (string).
//   fb_blink_diagnos_1: The function block BLINK generates a pulsating signal.The input consists of ENABLE of the type BOOL, as well as TIMELOW and TIMEHIGH of the type TIME.
//   axisdata[1].Axis_Inbb: A-0-0021.13 -RD- Axis is ready for power to the amplifier (bb)
//   FP_S_0_0095: Diagnostic message
//   drive1: Real axis "Drive1" with axis number 1
fb_blink_diagnos_1(ENABLE := axisdata[1].Axis_Inbb, TIMELOW := t#1s, TIMEHIGH := t#1s); // BLINK
fb_diagnose_1(
    Execute := fb_blink_diagnos_1.OUT,
    ParameterNumber := FP_S_0_0095,
    Axis := drive1,
    Value => str_diagnose_1); // MB_ReadStringParameter

// NETWORK 10
//   axisdata[2].Axis_Inbb: A-0-0021.13 -RD- Axis is ready for power to the amplifier (bb)
//   FP_S_0_0095: Diagnostic message
//   drive2: Real axis "Drive2" with axis number 2
fb_blink_diagnos_2(ENABLE := axisdata[2].Axis_Inbb, TIMELOW := t#1s, TIMEHIGH := t#1s); // BLINK
fb_diagnose_2(
    Execute := fb_blink_diagnos_2.OUT,
    ParameterNumber := FP_S_0_0095,
    Axis := drive2,
    Value => str_diagnose_2); // MB_ReadStringParameter

// NETWORK 11
//   axisdata[3].Axis_Inbb: A-0-0021.13 -RD- Axis is ready for power to the amplifier (bb)
//   FP_S_0_0095: Diagnostic message
//   drive3: Real axis "Drive3" with axis number 3
fb_blink_diagnos_3(ENABLE := axisdata[3].Axis_Inbb, TIMELOW := t#1s, TIMEHIGH := t#1s); // BLINK
fb_diagnose_3(
    Execute := fb_blink_diagnos_3.OUT,
    ParameterNumber := FP_S_0_0095,
    Axis := drive3,
    Value => str_diagnose_3); // MB_ReadStringParameter

// NETWORK 12 (disabled)
//   axisdata[4].Axis_Inbb: A-0-0021.13 -RD- Axis is ready for power to the amplifier (bb)
//   FP_S_0_0095: Diagnostic message
//   drive4: Real axis "Drive4" with axis number 4
// fb_blink_diagnos_4(ENABLE := axisdata[4].Axis_Inbb, TIMELOW := t#1s, TIMEHIGH := t#1s); // BLINK
// fb_diagnose_4(
//     Execute := fb_blink_diagnos_4.OUT,
//     ParameterNumber := FP_S_0_0095,
//     Axis := drive4,
//     Value => str_diagnose_4); // MB_ReadStringParameter

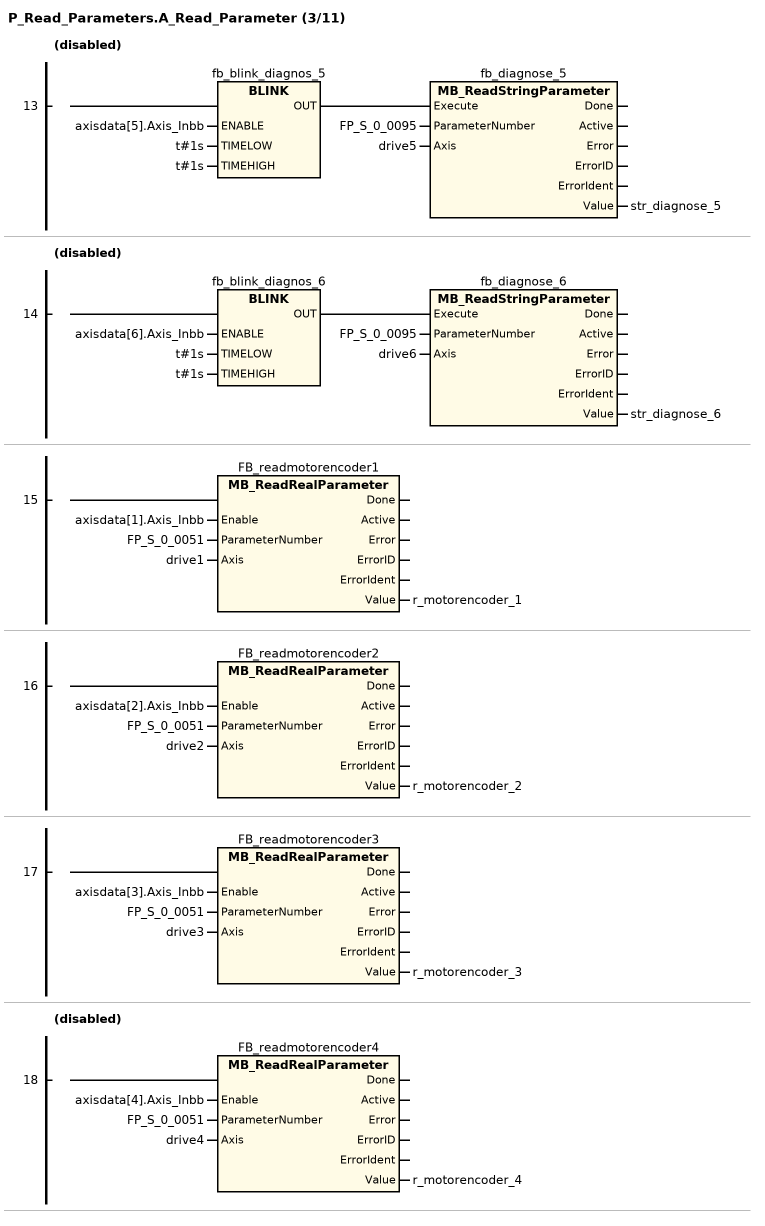
// NETWORK 13 (disabled)
//   axisdata[5].Axis_Inbb: A-0-0021.13 -RD- Axis is ready for power to the amplifier (bb)
//   FP_S_0_0095: Diagnostic message
//   drive5: Real axis "Drive5" with axis number 5
// fb_blink_diagnos_5(ENABLE := axisdata[5].Axis_Inbb, TIMELOW := t#1s, TIMEHIGH := t#1s); // BLINK
// fb_diagnose_5(
//     Execute := fb_blink_diagnos_5.OUT,
//     ParameterNumber := FP_S_0_0095,
//     Axis := drive5,
//     Value => str_diagnose_5); // MB_ReadStringParameter

// NETWORK 14 (disabled)
//   axisdata[6].Axis_Inbb: A-0-0021.13 -RD- Axis is ready for power to the amplifier (bb)
//   FP_S_0_0095: Diagnostic message
//   drive6: Real axis "Drive6" with axis number 6
// fb_blink_diagnos_6(ENABLE := axisdata[6].Axis_Inbb, TIMELOW := t#1s, TIMEHIGH := t#1s); // BLINK
// fb_diagnose_6(
//     Execute := fb_blink_diagnos_6.OUT,
//     ParameterNumber := FP_S_0_0095,
//     Axis := drive6,
//     Value => str_diagnose_6); // MB_ReadStringParameter

// NETWORK 15
//   axisdata[1].Axis_Inbb: A-0-0021.13 -RD- Axis is ready for power to the amplifier (bb)
//   FP_S_0_0051: Position feedback value 1
//   drive1: Real axis "Drive1" with axis number 1
FB_readmotorencoder1(
    Enable := axisdata[1].Axis_Inbb,
    ParameterNumber := FP_S_0_0051,
    Axis := drive1,
    Value => r_motorencoder_1); // MB_ReadRealParameter

// NETWORK 16
//   axisdata[2].Axis_Inbb: A-0-0021.13 -RD- Axis is ready for power to the amplifier (bb)
//   FP_S_0_0051: Position feedback value 1
//   drive2: Real axis "Drive2" with axis number 2
FB_readmotorencoder2(
    Enable := axisdata[2].Axis_Inbb,
    ParameterNumber := FP_S_0_0051,
    Axis := drive2,
    Value => r_motorencoder_2); // MB_ReadRealParameter

// NETWORK 17
//   axisdata[3].Axis_Inbb: A-0-0021.13 -RD- Axis is ready for power to the amplifier (bb)
//   FP_S_0_0051: Position feedback value 1
//   drive3: Real axis "Drive3" with axis number 3
FB_readmotorencoder3(
    Enable := axisdata[3].Axis_Inbb,
    ParameterNumber := FP_S_0_0051,
    Axis := drive3,
    Value => r_motorencoder_3); // MB_ReadRealParameter

// NETWORK 18 (disabled)
//   axisdata[4].Axis_Inbb: A-0-0021.13 -RD- Axis is ready for power to the amplifier (bb)
//   FP_S_0_0051: Position feedback value 1
//   drive4: Real axis "Drive4" with axis number 4
// FB_readmotorencoder4(
//     Enable := axisdata[4].Axis_Inbb,
//     ParameterNumber := FP_S_0_0051,
//     Axis := drive4,
//     Value => r_motorencoder_4); // MB_ReadRealParameter

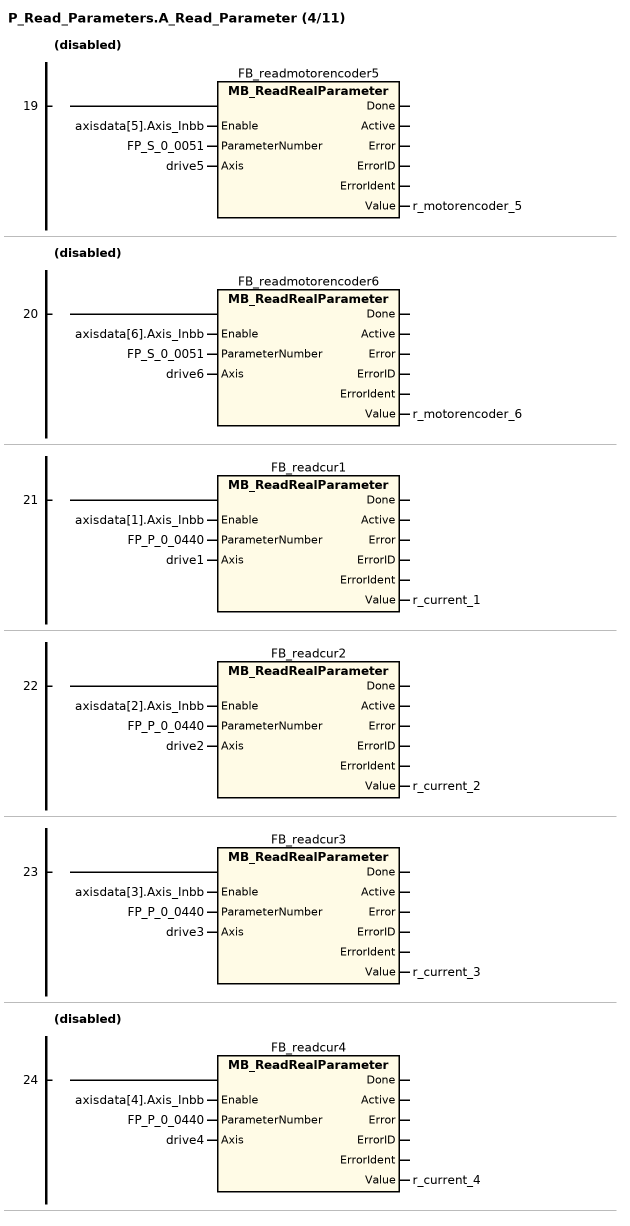
// NETWORK 19 (disabled)
//   axisdata[5].Axis_Inbb: A-0-0021.13 -RD- Axis is ready for power to the amplifier (bb)
//   FP_S_0_0051: Position feedback value 1
//   drive5: Real axis "Drive5" with axis number 5
// FB_readmotorencoder5(
//     Enable := axisdata[5].Axis_Inbb,
//     ParameterNumber := FP_S_0_0051,
//     Axis := drive5,
//     Value => r_motorencoder_5); // MB_ReadRealParameter

// NETWORK 20 (disabled)
//   axisdata[6].Axis_Inbb: A-0-0021.13 -RD- Axis is ready for power to the amplifier (bb)
//   FP_S_0_0051: Position feedback value 1
//   drive6: Real axis "Drive6" with axis number 6
// FB_readmotorencoder6(
//     Enable := axisdata[6].Axis_Inbb,
//     ParameterNumber := FP_S_0_0051,
//     Axis := drive6,
//     Value => r_motorencoder_6); // MB_ReadRealParameter

// NETWORK 21
//   FB_readcur1: With the function block "MB_ReadRealParameter" it is possible to read the current value of a parameter. The return value is REAL.
//   axisdata[1].Axis_Inbb: A-0-0021.13 -RD- Axis is ready for power to the amplifier (bb)
//   FP_P_0_0440: Actual output current value (absolute value)
//   drive1: Real axis "Drive1" with axis number 1
//   r_current_1: FP_P_0_0440,Actual output current value absolute value
FB_readcur1(
    Enable := axisdata[1].Axis_Inbb,
    ParameterNumber := FP_P_0_0440,
    Axis := drive1,
    Value => r_current_1); // MB_ReadRealParameter

// NETWORK 22
//   axisdata[2].Axis_Inbb: A-0-0021.13 -RD- Axis is ready for power to the amplifier (bb)
//   FP_P_0_0440: Actual output current value (absolute value)
//   drive2: Real axis "Drive2" with axis number 2
FB_readcur2(
    Enable := axisdata[2].Axis_Inbb,
    ParameterNumber := FP_P_0_0440,
    Axis := drive2,
    Value => r_current_2); // MB_ReadRealParameter

// NETWORK 23
//   axisdata[3].Axis_Inbb: A-0-0021.13 -RD- Axis is ready for power to the amplifier (bb)
//   FP_P_0_0440: Actual output current value (absolute value)
//   drive3: Real axis "Drive3" with axis number 3
FB_readcur3(
    Enable := axisdata[3].Axis_Inbb,
    ParameterNumber := FP_P_0_0440,
    Axis := drive3,
    Value => r_current_3); // MB_ReadRealParameter

// NETWORK 24 (disabled)
//   axisdata[4].Axis_Inbb: A-0-0021.13 -RD- Axis is ready for power to the amplifier (bb)
//   FP_P_0_0440: Actual output current value (absolute value)
//   drive4: Real axis "Drive4" with axis number 4
// FB_readcur4(
//     Enable := axisdata[4].Axis_Inbb,
//     ParameterNumber := FP_P_0_0440,
//     Axis := drive4,
//     Value => r_current_4); // MB_ReadRealParameter

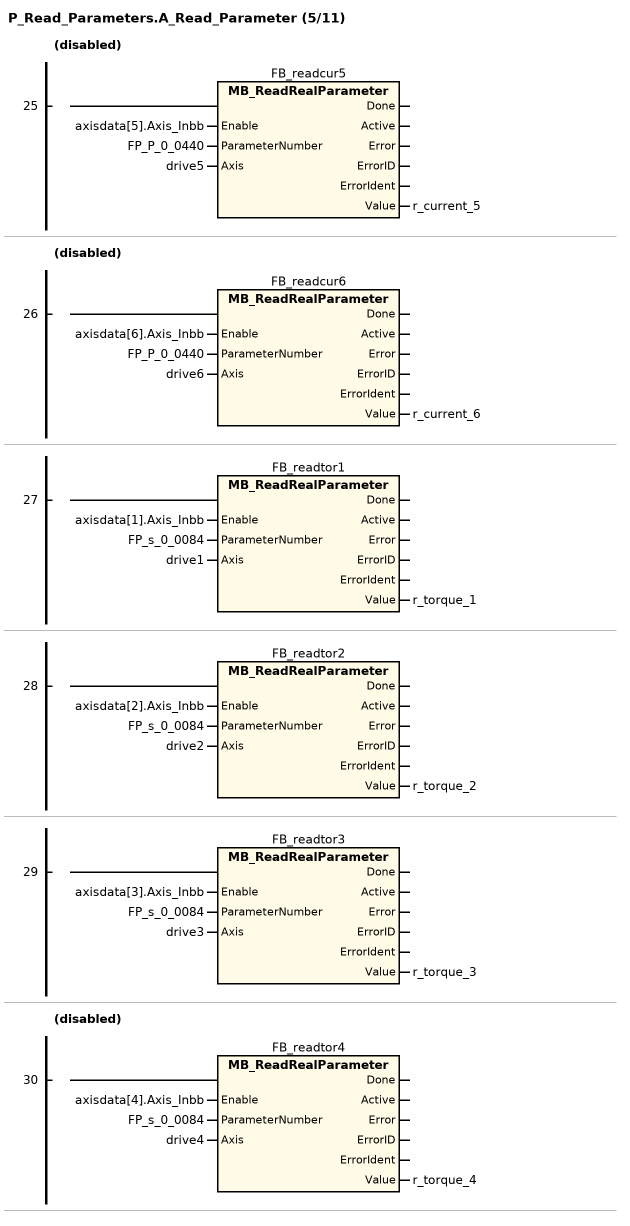
// NETWORK 25 (disabled)
//   axisdata[5].Axis_Inbb: A-0-0021.13 -RD- Axis is ready for power to the amplifier (bb)
//   FP_P_0_0440: Actual output current value (absolute value)
//   drive5: Real axis "Drive5" with axis number 5
// FB_readcur5(
//     Enable := axisdata[5].Axis_Inbb,
//     ParameterNumber := FP_P_0_0440,
//     Axis := drive5,
//     Value => r_current_5); // MB_ReadRealParameter

// NETWORK 26 (disabled)
//   axisdata[6].Axis_Inbb: A-0-0021.13 -RD- Axis is ready for power to the amplifier (bb)
//   FP_P_0_0440: Actual output current value (absolute value)
//   drive6: Real axis "Drive6" with axis number 6
// FB_readcur6(
//     Enable := axisdata[6].Axis_Inbb,
//     ParameterNumber := FP_P_0_0440,
//     Axis := drive6,
//     Value => r_current_6); // MB_ReadRealParameter

// NETWORK 27
//   axisdata[1].Axis_Inbb: A-0-0021.13 -RD- Axis is ready for power to the amplifier (bb)
//   FP_s_0_0084: Torque/force feedback value
//   drive1: Real axis "Drive1" with axis number 1
//   r_torque_1: FP_S_0_0084,Torque force feedback value
FB_readtor1(
    Enable := axisdata[1].Axis_Inbb,
    ParameterNumber := FP_s_0_0084,
    Axis := drive1,
    Value => r_torque_1); // MB_ReadRealParameter

// NETWORK 28
//   axisdata[2].Axis_Inbb: A-0-0021.13 -RD- Axis is ready for power to the amplifier (bb)
//   FP_s_0_0084: Torque/force feedback value
//   drive2: Real axis "Drive2" with axis number 2
FB_readtor2(
    Enable := axisdata[2].Axis_Inbb,
    ParameterNumber := FP_s_0_0084,
    Axis := drive2,
    Value => r_torque_2); // MB_ReadRealParameter

// NETWORK 29
//   axisdata[3].Axis_Inbb: A-0-0021.13 -RD- Axis is ready for power to the amplifier (bb)
//   FP_s_0_0084: Torque/force feedback value
//   drive3: Real axis "Drive3" with axis number 3
FB_readtor3(
    Enable := axisdata[3].Axis_Inbb,
    ParameterNumber := FP_s_0_0084,
    Axis := drive3,
    Value => r_torque_3); // MB_ReadRealParameter

// NETWORK 30 (disabled)
//   axisdata[4].Axis_Inbb: A-0-0021.13 -RD- Axis is ready for power to the amplifier (bb)
//   FP_s_0_0084: Torque/force feedback value
//   drive4: Real axis "Drive4" with axis number 4
// FB_readtor4(
//     Enable := axisdata[4].Axis_Inbb,
//     ParameterNumber := FP_s_0_0084,
//     Axis := drive4,
//     Value => r_torque_4); // MB_ReadRealParameter

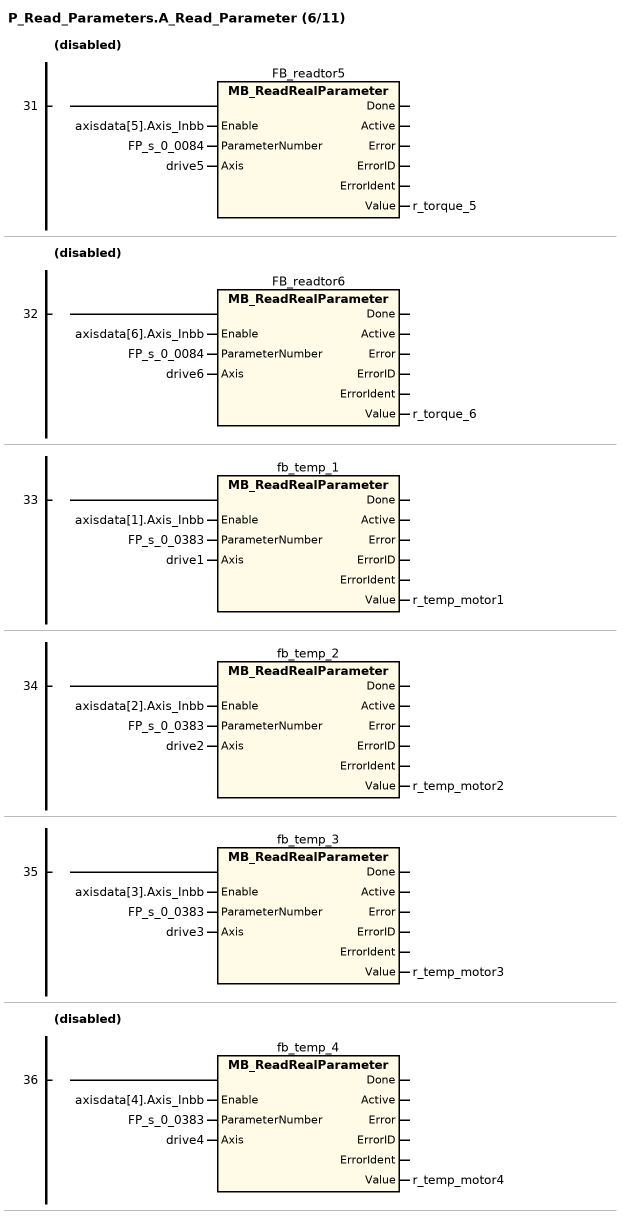
// NETWORK 31 (disabled)
//   axisdata[5].Axis_Inbb: A-0-0021.13 -RD- Axis is ready for power to the amplifier (bb)
//   FP_s_0_0084: Torque/force feedback value
//   drive5: Real axis "Drive5" with axis number 5
// FB_readtor5(
//     Enable := axisdata[5].Axis_Inbb,
//     ParameterNumber := FP_s_0_0084,
//     Axis := drive5,
//     Value => r_torque_5); // MB_ReadRealParameter

// NETWORK 32 (disabled)
//   axisdata[6].Axis_Inbb: A-0-0021.13 -RD- Axis is ready for power to the amplifier (bb)
//   FP_s_0_0084: Torque/force feedback value
//   drive6: Real axis "Drive6" with axis number 6
// FB_readtor6(
//     Enable := axisdata[6].Axis_Inbb,
//     ParameterNumber := FP_s_0_0084,
//     Axis := drive6,
//     Value => r_torque_6); // MB_ReadRealParameter

// NETWORK 33
//   axisdata[1].Axis_Inbb: A-0-0021.13 -RD- Axis is ready for power to the amplifier (bb)
//   FP_s_0_0383: Motor temperature
//   drive1: Real axis "Drive1" with axis number 1
//   r_temp_motor1: FP_S_0_0383,Motor temperature
fb_temp_1(
    Enable := axisdata[1].Axis_Inbb,
    ParameterNumber := FP_s_0_0383,
    Axis := drive1,
    Value => r_temp_motor1); // MB_ReadRealParameter

// NETWORK 34
//   axisdata[2].Axis_Inbb: A-0-0021.13 -RD- Axis is ready for power to the amplifier (bb)
//   FP_s_0_0383: Motor temperature
//   drive2: Real axis "Drive2" with axis number 2
fb_temp_2(
    Enable := axisdata[2].Axis_Inbb,
    ParameterNumber := FP_s_0_0383,
    Axis := drive2,
    Value => r_temp_motor2); // MB_ReadRealParameter

// NETWORK 35
//   axisdata[3].Axis_Inbb: A-0-0021.13 -RD- Axis is ready for power to the amplifier (bb)
//   FP_s_0_0383: Motor temperature
//   drive3: Real axis "Drive3" with axis number 3
fb_temp_3(
    Enable := axisdata[3].Axis_Inbb,
    ParameterNumber := FP_s_0_0383,
    Axis := drive3,
    Value => r_temp_motor3); // MB_ReadRealParameter

// NETWORK 36 (disabled)
//   axisdata[4].Axis_Inbb: A-0-0021.13 -RD- Axis is ready for power to the amplifier (bb)
//   FP_s_0_0383: Motor temperature
//   drive4: Real axis "Drive4" with axis number 4
// fb_temp_4(
//     Enable := axisdata[4].Axis_Inbb,
//     ParameterNumber := FP_s_0_0383,
//     Axis := drive4,
//     Value => r_temp_motor4); // MB_ReadRealParameter

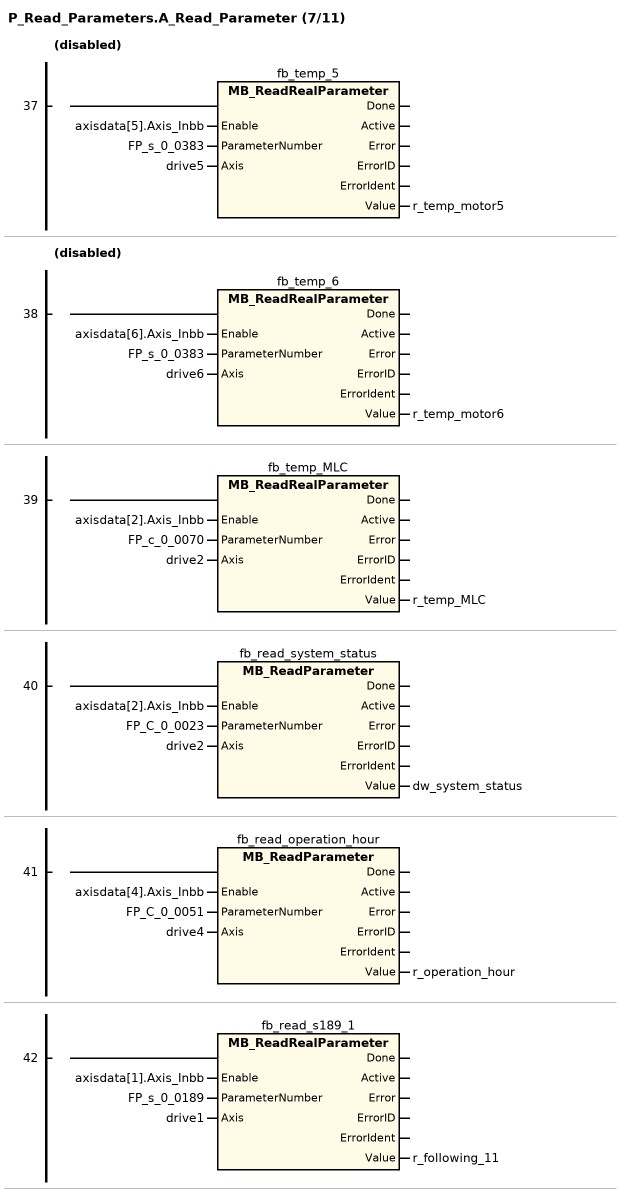
// NETWORK 37 (disabled)
//   axisdata[5].Axis_Inbb: A-0-0021.13 -RD- Axis is ready for power to the amplifier (bb)
//   FP_s_0_0383: Motor temperature
//   drive5: Real axis "Drive5" with axis number 5
// fb_temp_5(
//     Enable := axisdata[5].Axis_Inbb,
//     ParameterNumber := FP_s_0_0383,
//     Axis := drive5,
//     Value => r_temp_motor5); // MB_ReadRealParameter

// NETWORK 38 (disabled)
//   axisdata[6].Axis_Inbb: A-0-0021.13 -RD- Axis is ready for power to the amplifier (bb)
//   FP_s_0_0383: Motor temperature
//   drive6: Real axis "Drive6" with axis number 6
// fb_temp_6(
//     Enable := axisdata[6].Axis_Inbb,
//     ParameterNumber := FP_s_0_0383,
//     Axis := drive6,
//     Value => r_temp_motor6); // MB_ReadRealParameter

// NETWORK 39
//   fb_temp_MLC: <<<<<<<<<<<<<<<<<<<<<<<<<<<<<<<<<<<<<<<add MLC temperature and operation hour(20100708)>>>>>>>>>>>>>>>>>>>>>>>>>>>>>>>>>>>>>
//   axisdata[2].Axis_Inbb: A-0-0021.13 -RD- Axis is ready for power to the amplifier (bb)
//   FP_c_0_0070: Control temperature
//   drive2: Real axis "Drive2" with axis number 2
//   r_temp_MLC: FP_c_0_0070,Control unit temperature
fb_temp_MLC(
    Enable := axisdata[2].Axis_Inbb,
    ParameterNumber := FP_c_0_0070,
    Axis := drive2,
    Value => r_temp_MLC); // MB_ReadRealParameter

// NETWORK 40
//   axisdata[2].Axis_Inbb: A-0-0021.13 -RD- Axis is ready for power to the amplifier (bb)
//   FP_C_0_0023: System status
//   drive2: Real axis "Drive2" with axis number 2
//   dw_system_status: FP_C_0_0023,MC system status,used for temperature warning
fb_read_system_status(
    Enable := axisdata[2].Axis_Inbb,
    ParameterNumber := FP_C_0_0023,
    Axis := drive2,
    Value => dw_system_status); // MB_ReadParameter

